WHILE (last-first)>1 DO
	first:=getNextFirstValid(first);
	last:=getNextLastValid(last);
	IF (first<0) OR (last<0) THEN
		RETURN;
	END_IF
END_WHILE

medianValue:=TRUE;
value:=	(inputs[first].input.value+inputs[last].input.value)/2;
END_METHOD

METHOD PRIVATE minValue : BOOL
VAR_INPUT
END_VAR
VAR_OUTPUT
	value:REAL;
END_VAR
VAR
	i:INT;
END_VAR
value:=RNaN();

FOR i:=0 TO arrayMaxIndex DO
	IF isValidInput(inputs[i]) THEN
		IF (FPU.IsRealNaN(value) OR (inputs[i].input.value < value)) THEN
			value:= inputs[i].input.value;
			minValue:=TRUE;
		END_IF
	END_IF
END_FOR
END_METHOD

METHOD PRIVATE compare:bool
VAR_INPUT
	nas1: AnalogItem;
	nas2: AnalogItem;
END_VAR
IF (__ISVALIDREF(nas1.input) AND (NOT __ISVALIDREF (nas2.input))) THEN
	compare:=FALSE;
	RETURN;
END_IF

IF (NOT __ISVALIDREF(nas1.input) AND (__ISVALIDREF (nas2.input))) THEN
	compare:=TRUE;
	RETURN;
END_IF

compare:=FALSE;

IF (__ISVALIDREF(nas1.input) AND __ISVALIDREF (nas2.input)) THEN
	IF 	(nas1.input.interval>=statusAi.normal)AND(nas2.input.interval>=statusAi.normal) THEN
		compare:=nas1.input.value>nas2.input.value;
	ELSE
		compare:=(nas1.input.interval<statusAi.normal)AND(nas2.input.interval>=statusAi.normal)	;			
	END_IF
END_IF
END_METHOD

METHOD sort
VAR_INPUT
END_VAR
VAR
	i,j:INT;
	item:AnalogItem;
	compareResult:BOOL;
END_VAR
FOR i:=1 TO arrayMaxIndex DO
	item:= inputs[i];  
	j:= i - 1;
	compareResult:=compare(nas1:=inputs[j],nas2:=item);
	WHILE (j >= 0) AND (compareResult) DO    
	   	inputs[j + 1]:= inputs[j];
	 	j:=j-1;
	 	IF j>=0 THEN
			compareResult:=compare(nas1:=inputs[j],nas2:=item);
		END_IF
	END_WHILE;
	inputs[j + 1]:= item;
END_FOR
END_METHOD

METHOD PROTECTED writePersistent
VAR_INPUT
END_VAR
SUPER^.writePersistent();
writeValue(value:=FPU.RealToStr(maxDelta),comment:='MAX разброс');
END_METHOD

END_FUNCTION_BLOCK

// lowLevel_ecl/kontroller/mlp/Sources/AoSourceMlp
{attribute 'symbol' := 'none'}
FUNCTION_BLOCK PUBLIC AoSourceMlp EXTENDS AOSource
IMPLEMENTS IMlpSource;
VAR_INPUT
	outLL:REAL:=4000;
	outHl:REAL:=20000;
END_VAR
VAR_OUTPUT
END_VAR
VAR
	elpk:REFERENCE TO Elpk04;
END_VAR

SUPER^();

METHOD setKontroller
VAR_INPUT
	nKontroller	: REFERENCE TO Elpk04;
END_VAR
elpk REF=nKontroller;
END_METHOD

METHOD PROTECTED writeData
VAR_INPUT
	val:REAL;
END_VAR
IF (HL<>LL) THEN
	elpk.Aout_[addr]:=(val-Ll)*(outHl-outLL)/(Hl-Ll)+outLL;
END_IF
END_METHOD

END_FUNCTION_BLOCK

// lowLevel_ecl/kontroller/mlp/Sources/AiFrequenceMlp
{attribute 'symbol' := 'none'}
FUNCTION_BLOCK AiFrequenceMlp EXTENDS AISource
IMPLEMENTS IMlpSource;
VAR_INPUT
	dK:REAL:=1;
	dB:REAL:=0;
END_VAR
VAR_OUTPUT
	{attribute 'symbol' := 'read'}
	k:REAL;
	{attribute 'symbol' := 'read'}
	b:REAL;
END_VAR
VAR
	elpk:REFERENCE TO Elpk04;
	source:AnalogRecalc;
	
	{attribute 'symbol' := 'readwrite'}
	newk:REAL;
	{attribute 'symbol' := 'readwrite'}
	newb:REAL;
END_VAR

SUPER^();

METHOD PROTECTED readPersistent
VAR_INPUT
END_VAR
SUPER^.readPersistent();
K:=FPU.StrToReal(readValue());
B:=FPU.StrToReal(readValue());
END_METHOD

METHOD setKontroller
VAR_INPUT
	nKontroller	: REFERENCE TO Elpk04;
END_VAR
elpk REF=nKontroller;
END_METHOD

METHOD PROTECTED GetData : Real
VAR_INPUT
END_VAR
VAR_OUTPUT
	o_interval:statusAi;
END_VAR
source.input:=elpk.AIn_[addr].val;
source.k:=K;
source.b:=B;
source.h:=histeresis;
source.ap:=aperturFilter;
source.dp:=pikFiler;
source.ds:=exponentialFilter;
source.de:=rassoglasovanie;
source();

GetData:=source.value;

o_interval:=statusAi.normal;
END_METHOD

METHOD PROTECTED writePersistent
VAR_INPUT
END_VAR
SUPER^.writePersistent();
writeValue(value:=FPU.RealToStr(k),comment:='k');
writeValue(value:=FPU.RealToStr(b),comment:='b');
END_METHOD

METHOD PROTECTED setDefaultPersistent:BOOL
VAR_INPUT
END_VAR
SUPER^.setDefaultPersistent();
k:=dK;
b:=dB;
setDefaultPersistent:=TRUE;
END_METHOD

END_FUNCTION_BLOCK

// lowLevel_ecl/kontroller/mlp/Sources/DiSourceMlp
{attribute 'symbol' := 'none'}
FUNCTION_BLOCK DiSourceMlp EXTENDS DISource
IMPLEMENTS IMlpSource;
VAR_INPUT
END_VAR
VAR_OUTPUT
END_VAR
VAR
	elpk:REFERENCE TO Elpk04;
	bitNumber:int;
END_VAR

SUPER^();

METHOD setKontroller
VAR_INPUT
	nKontroller	: REFERENCE TO Elpk04;
END_VAR
elpk REF=nKontroller;
END_METHOD

METHOD PROTECTED getData : word
VAR_INPUT
END_VAR
VAR_OUTPUT
	reliability:WORD;
END_VAR
VAR
	_value:WORD;
	_reliability:BOOL;
END_VAR

_value:=elpk.DIn_[addr].val;
FOR bitNumber:=0 TO 7 DO
	_reliability:=UINT_TO_BOOL(SHR (_value, bitNumber*2) AND 16#2);
	reliability:=reliability OR SHL(BOOL_TO_WORD(_reliability),bitNumber);
	IF _reliability THEN
		getData:=getData OR SHL(SHR (_value, bitNumber*2) AND 16#1,bitNumber);
	END_IF;
END_FOR
END_METHOD

END_FUNCTION_BLOCK

// lowLevel_ecl/kontroller/mlp/Sources/AnalogDiSourceMlp
	{attribute 'symbol' := 'none'}
FUNCTION_BLOCK AnalogDiSourceMlp EXTENDS CustomSource
IMPLEMENTS IMlpSource;
VAR_INPUT
	addr:BYTE;
		 	{attribute 'symbol' := 'readwrite'}
	newTrueLow:REAL;
		 	{attribute 'symbol' := 'readwrite'}
	newTrueHigh:REAL;
		 	{attribute 'symbol' := 'readwrite'}
	newFalseLow:REAL;
		 	{attribute 'symbol' := 'readwrite'}
	newFalseHigh:REAL;
END_VAR
VAR_OUTPUT
	Q:InversableReliableBit;
	{attribute 'symbol' := 'readwrite'}
	value:REAL;
	{attribute 'symbol' := 'readwrite'}
	interval:statusAi;
END_VAR
VAR
	elpk:REFERENCE TO Elpk04;
	source:AnalogRecalc;
		 	{attribute 'symbol' := 'read'}
	trueLow:REAL;
		 	{attribute 'symbol' := 'read'}
	trueHigh:REAL;
		 	{attribute 'symbol' := 'read'}
	falseLow:REAL;
		 	{attribute 'symbol' := 'read'}
	falseHigh:REAL;
END_VAR
VAR CONSTANT
		cmd_changeLimits:WORD:=1;
END_VAR

SUPER^();

IF NOT imit THEN
	source.k:=0.001;
	source.input:=elpk.AIn_[addr].val;
	source();
	value:=source.value;
END_IF

resetCommand();

IF (value>=4) AND (value<=20)  THEN
	IF (value>=falseLow) AND (value<=falseHigh) THEN
		Q.setReliability(TRUE);
		Q.setValue(FALSE);
	ELSIF (value>=trueLow) AND (value<=trueHigh) THEN
		Q.setReliability(TRUE);
		Q.setValue(TRUE);
	ELSE
		Q.setReliability(FALSE);
	END_IF
ELSE
	Q.setReliability(FALSE);
END_IF

METHOD PROTECTED readPersistent
VAR_INPUT
END_VAR
trueLow:=FPU.StrToReal(readValue());
trueHigh:=FPU.StrToReal(readValue());
falseLow:=FPU.StrToReal(readValue());
falseHigh:=FPU.StrToReal(readValue());
END_METHOD

METHOD PROTECTED writePersistent
VAR_INPUT
END_VAR
writeValue(value:=FPU.RealToStr(trueLow),comment:='trueLow');
writeValue(value:=FPU.RealToStr(trueHigh),comment:='trueHigh');
writeValue(value:=FPU.RealToStr(falseLow),comment:='falseLow');
writeValue(value:=FPU.RealToStr(falseHigh),comment:='falseHigh');
END_METHOD

METHOD setLimits
VAR_INPUT
	nFalseLow:REAL;
	nFalseHigh:REAL;
	nTrueLow:REAL;
	nTrueHigh:REAL;

END_VAR
setCmd(nCmd:=cmd_ChangeLimits);
falseLow:=nFalseLow;
falseHigh:=nFalseHigh;
trueLow:=nTrueLow;
trueHigh:=nTrueHigh;

SaveToFile();
END_METHOD

METHOD PROTECTED processCmd;
VAR_INPUT
	cmd:UINT;
	sender:UINT;
	parametr:UINT;
END_VAR
CASE cmd OF
	cmd_changeLimits:setLimits(nFalseLow:=newFalseLow,nFalseHigh:=newFalseHigh,nTrueLow:=newTrueLow,nTrueHigh:=newTrueHigh);
END_CASE
END_METHOD

METHOD setKontroller
VAR_INPUT
	nKontroller	: REFERENCE TO Elpk04;
END_VAR
elpk REF=nKontroller;
END_METHOD

END_FUNCTION_BLOCK

// lowLevel_ecl/kontroller/baseSources/CustomSource
	{attribute 'symbol' := 'none'}
FUNCTION_BLOCK CustomSource EXTENDS BaseIm
IMPLEMENTS ISource
VAR_INPUT

END_VAR
VAR_OUTPUT

END_VAR
VAR
	_imit:BOOL;  
END_VAR

SUPER^();

{attribute 'symbol' := 'none'}
PROPERTY imit : BOOL
SET
_imit:=imit;
END_SET
GET
imit:=_imit;
END_GET
END_PROPERTY

END_FUNCTION_BLOCK

// lowLevel_ecl/kontroller/mlp/Sources/AiSourceMlp
{attribute 'symbol' := 'none'}
FUNCTION_BLOCK AiSourceMlp EXTENDS AISource
IMPLEMENTS IMlpSource;
VAR_INPUT
	inpLL:REAL:=4000;
	inpHl:REAL:=20000;
END_VAR
VAR_OUTPUT
END_VAR
VAR
	elpk:REFERENCE TO Elpk04;
	source:AnalogRecalc;
END_VAR

SUPER^();

METHOD setKontroller
VAR_INPUT
	nKontroller	: REFERENCE TO Elpk04;
END_VAR
elpk REF=nKontroller;
END_METHOD

METHOD PROTECTED GetData : Real
VAR_INPUT
END_VAR
VAR_OUTPUT
	o_interval:statusAi;
END_VAR
source.input:=elpk.AIn_[addr].val;
source.k:=(HL-LL)/(inpHl-inpLL);
source.b:=LL-source.k*inpLL;

source.h:=histeresis;
source.ap:=aperturFilter;
source.dp:=pikFiler;
source.ds:=exponentialFilter;
source.de:=rassoglasovanie;
source();

GetData:=source.value;

IF (NOT (elpk.AIn_[addr].f.0)) OR (NOT (elpk.AIn_[addr].f.2)) OR  (elpk.AIn_[addr].f.1) THEN
	 o_interval:=statusAi.NOTDEFINED;
ELSE
	o_interval:=statusAi.normal;	
END_IF
END_METHOD

END_FUNCTION_BLOCK

// lowLevel_ecl/kontroller/mlp/Sources/DoSourceMlp
{attribute 'symbol' := 'none'}
FUNCTION_BLOCK DoSourceMlp EXTENDS DOSource
IMPLEMENTS IMlpSource;
VAR_INPUT
END_VAR
VAR_OUTPUT
END_VAR
VAR
	elpk:REFERENCE TO Elpk04;
END_VAR

SUPER^();

METHOD setKontroller
VAR_INPUT
	nKontroller	: REFERENCE TO Elpk04;
END_VAR
elpk REF=nKontroller;
END_METHOD

METHOD writeData
VAR_INPUT
	value:WORD;
END_VAR
elpk.Dout_[addr]:=value;
END_METHOD

END_FUNCTION_BLOCK

// lowLevel_ecl/im/extensions/ExtNarabotka
	{attribute 'symbol' := 'none'}
FUNCTION_BLOCK ExtNarabotka EXTENDS BaseObject
VAR_INPUT
	saveInterval:TIME:=T#30S;
END_VAR
VAR_OUTPUT
	{attribute 'symbol' := 'read'}
	narabotka:UDINT;	
END_VAR
VAR
END_VAR
VAR
	timer:RTC;	
	saveTimer:TON;
END_VAR

SUPER^();
timer();

IF timer.Q THEN
	narabotka:=DT_TO_UDINT( timer.CDT);
END_IF

saveTimer(IN:=TRUE,PT:=saveInterval);
IF saveTimer.Q THEN
	SaveToFile();
	saveTimer(IN:=FALSE);
END_IF

METHOD PROTECTED readPersistent
VAR_INPUT
END_VAR
narabotka:=STRING_TO_UDINT(readValue());
END_METHOD

METHOD PUBLIC reset
VAR_INPUT
END_VAR
timer.PDT:=UINT_TO_DT(0);
IF timer.EN THEN
	timer(EN:=FALSE);
	timer(EN:=TRUE);
END_IF
narabotka:=0;
END_METHOD

METHOD PUBLIC start
VAR_INPUT
END_VAR
timer.PDT:=UDINT_TO_DT(narabotka);
timer.EN:=TRUE;
END_METHOD

PROPERTY PUBLIC started : Bool
GET
started:=timer.Q;
END_GET
SET
IF started then
	IF NOT timer.Q THEN
		start();
	END_IF
ELSE
	IF timer.Q THEN
		stop();
	END_IF
END_IF
END_SET
END_PROPERTY

METHOD PUBLIC stop
VAR_INPUT
END_VAR
timer.EN:=FALSE;
SaveToFile();
END_METHOD

METHOD PROTECTED writePersistent
VAR_INPUT
END_VAR
writeValue(value:= UDINT_TO_STRING(narabotka),'Наработка');
END_METHOD

END_FUNCTION_BLOCK

// lowLevel_ecl/im/Mokveld/Mokveld
	{attribute 'symbol' := 'none'}
FUNCTION_BLOCK Mokveld EXTENDS BaseIm
VAR_INPUT
	inPosition:REFERENCE TO AISource;
	inAssignment:REFERENCE TO AOSource;
	
	dMaxOpenSpeed:REAL:=RNaN();
	dMaxCloseSpeed:REAL:=RNaN();
	
	maxPositionMismatch:REAL:=RNaN();
	posotionnMismatchDelay:TIME:=T#5S;
	
	openPosition:REAL:=95;
	closePosition:REAL:=5;
	
		{attribute 'symbol' := 'readwrite'}
	newTarget:REAL;
END_VAR
VAR_OUTPUT
	{attribute 'symbol' := 'read'}
	position:REAL;
	{attribute 'symbol' := 'read'}
	target:REAL;	

	Assignment:REAL;	
	
	onStatus:statusDualInput;
	
	positionMismatch:BOOL;
END_VAR
VAR
	maxOpenSpeed:REAL;
	maxCloseSpeed:REAL;
	lastCallTimer:Ton:=(pt:=T#1H);
	posotionErrorTimer:TON;
END_VAR
VAR CONSTANT
	cmd_setTarget:WORD:=1;
END_VAR
VAR_TEMP
	delta:REAL:=RNaN();
END_VAR

SUPER^();

IF __ISVALIDREF(inPosition) THEN
	position:=inPosition.value;
	
	IF inPosition.interval>=statusAi.normal THEN
		IF (NOT FPU.IsRealNaN(maxPositionMismatch)) AND __ISVALIDREF(inAssignment) THEN
			posotionErrorTimer(IN:= rABS(inAssignment.Value-inPosition.value)>maxPositionMismatch,PT:=posotionnMismatchDelay);
			PositionMismatch:=posotionErrorTimer.Q;
		END_IF	
		onStatus:=calcOnStatus();
	ELSE
		onStatus:=statusDualInput.STATUS_ERROR;
		posotionErrorTimer(IN:=FALSE);
	END_IF
ELSE
	IF __ISVALIDREF(inAssignment) THEN
		position:=inAssignment.Value;
		onStatus:=calcOnStatus();			
	END_IF
END_IF

IF __ISVALIDREF(inAssignment) THEN
	inAssignment.DisableOpcControl();

	lastCallTimer();
	IF (target>inAssignment.Value) THEN 
		IF NOT FPU.IsRealNaN(maxOpenSpeed) THEN 
			delta:=maxOpenSpeed*(TIME_TO_REAL(lastCallTimer.ET)/1000);
		END_IF;
	ELSE
		IF NOT FPU.IsRealNaN(maxCloseSpeed) THEN
			delta:=-maxCloseSpeed*(TIME_TO_REAL(lastCallTimer.ET)/1000);
		END_IF	
	END_IF
	lastCallTimer(in:=FALSE);
	lastCallTimer(in:=TRUE);
		
	IF (NOT FPU.IsRealNaN(delta)) AND (ABS(delta)<ABS(inAssignment.Value-target)) THEN
		Assignment:=inAssignment.Value+delta;
	ELSE
		Assignment:=target;	
	END_IF
	
	inAssignment.setValue(nValue:=Assignment);
END_IF

METHOD PROTECTED calcOnStatus: statusDualInput
VAR_INPUT
END_VAR
IF (position<closePosition) THEN
	calcOnStatus:=statusDualInput.STATUS_OFF;
ELSIF (position>openPosition) THEN
	calcOnStatus:=statusDualInput.STATUS_ON;
ELSE
	calcOnStatus:=statusDualInput.STATUS_TRANSITIONAL;
END_IF
END_METHOD

METHOD PRIVATE cmdSetTarget
VAR_INPUT
	nTarget:REAL;
END_VAR
setCmd(nCmd:=cmd_setTarget);
setTarget(nTarget:=nTarget);
resetCommand();
END_METHOD

METHOD PROTECTED processCmd;
VAR_INPUT
	cmd:UINT;
	sender:UINT;
	parametr:UINT;
END_VAR
SUPER^.processCmd(cmd,sender,parametr);
CASE cmd OF
	cmd_setTarget: cmdSetTarget(nTarget:=newTarget);
END_CASE
END_METHOD

METHOD PROTECTED readPersistent
VAR_INPUT
END_VAR
SUPER^.readPersistent();
maxOpenSpeed:=FPU.StrToReal(readValue());
maxCloseSpeed:=FPU.StrToReal(readValue());
openPosition:=FPU.StrToReal(readValue());
closePosition:=FPU.StrToReal(readValue());
END_METHOD

METHOD PROTECTED setDefaultPersistent:BOOL
VAR_INPUT
END_VAR
SUPER^.setDefaultPersistent();
maxOpenSpeed:=dMaxOpenSpeed;
maxCloseSpeed:=dMaxCloseSpeed;
setDefaultPersistent:=TRUE;
END_METHOD

METHOD PUBLIC setTarget
VAR_INPUT
	nTarget:REAL;
END_VAR
target:=nTarget;
END_METHOD

METHOD PUBLIC writeImStatus
VAR_INPUT
END_VAR
statusSet.setBits(0,2,onStatus);
statusSet.setBit(3,positionMismatch);
END_METHOD

METHOD PROTECTED writePersistent
VAR_INPUT
END_VAR
SUPER^.writePersistent();
writeValue(value:=FPU.RealToStr(maxOpenSpeed),comment:='maxOpenSpeed');
writeValue(value:=FPU.RealToStr(maxCloseSpeed),comment:='maxCloseSpeed');
writeValue(value:=FPU.RealToStr(openPosition),comment:='openPosition');
writeValue(value:=FPU.RealToStr(closePosition),comment:='closePosition');
END_METHOD

END_FUNCTION_BLOCK

// REZERV1/ADDCRC16
FUNCTION ADDCRC16 : WORD
VAR_INPUT
	X:BYTE;
	_CRC16T:WORD;
END_VAR
VAR
	CRC16_B:BOOL;
	I:INT;
	T:WORD;
END_VAR

FOR I:=1 TO 8 DO
	
	T:=BYTE_TO_WORD(X) XOR _CRC16T;
	IF (T AND 16#1) = 1// если нечетное, то = true
		THEN
		CRC16_B:=TRUE;
		ELSE
		CRC16_B:=FALSE;
	END_IF

	_CRC16T:= SHR(_CRC16T, 1);
	X:= SHR(X,1);
	IF CRC16_B THEN _CRC16T:=_CRC16T XOR 16#A001; END_IF;

END_FOR
ADDCRC16:=_CRC16T;

END_FUNCTION

// REZERV1/COM_Rd
FUNCTION_BLOCK COM_Rd
VAR CONSTANT
	Buff_size12:INT:=12;
	Byte_send12:UINT:=12;
END_VAR
VAR_INPUT
	PilaK_O:WORD;
	StatusK_O:WORD;
	ReadyK_O:WORD;
END_VAR
VAR_IN_OUT
//	IndexCmd:INT:=-1;// команда на запись переменной Index с экрана
	IndexCmd:INT;// команда на запись переменной Index с экрана - инициализировать сверху
	Cnt0:INT:=0;// счетчик правильных заголовков пакета: 0x81 + (длина=12) 
	Cnt100:INT:=0;// счетчик ошибок длины пакета 
	Cnt101:INT:=0;// счетчик ошибок признака начала пакета 0x81
	Cnt102:INT:=0;// счетчик ошибок CRC16
	Cnt3:INT:=0;// для ошибок Write
	Cnt21:INT:=0;// для ошибок Read
	Cnt22:INT:=0;// для ошибок Read
	Cnt23:INT:=0;// для ошибок Read
	Cnt24:INT:=0;// для ошибок Read
	Cnt25:INT:=0;// для ошибок Read
	Cnt26:INT:=0;// для ошибок Read
	Cnt27:INT:=0;// для ошибок Read
	Cnt28:INT:=0;// для ошибок Read
	Cnt29:INT:=0;// для ошибок Read
	Cnt30:INT:=0;// для ошибок Read
	Cnt31:INT:=0;// для ошибок Read
	Cnt32:INT:=0;// для ошибок Read
END_VAR
VAR_OUTPUT
	// принятое из соседнего
	PilaFromK:WORD;
	StatusFromK:WORD;
	ReadyFromK:WORD;
	ErrorCOM_Mess1, ErrorCOM_Mess2:WSTRING;
	
END_VAR
VAR
	Index:INT:=0;
//	IndexCmd:INT:=-1;// команда на запись переменной Index с экрана
	I1, I2, I3, I4 :INT;// переменные временного использования
	PP1, PP2, PP3, PP4, PP5 : RTS_IEC_RESULT;
///	H1 : RTS_IEC_HANDLE;// pointer to byte
///	S1 : Com_Settings;
///	S1ex : Com_SettingsEX;

{attribute 'displaymode':='hex'} 
	Buff : ARRAY[1..Buff_size12] OF BYTE;
{attribute 'displaymode':='hex'} 
	Buff2 : ARRAY[1..Buff_size12] OF BYTE;
//{attribute 'displaymode':='hex'} 
//	Buff22 : ARRAY[1..Buff_size12] OF BYTE;
//	ErrorCOM_Mess1, ErrorCOM_Mess2:WSTRING;
	
	
	WW1, WW2, WW3,WW4,WW5,WW6,WW7,WW8,WW9,WW10,WW10a,WW10b:UDINT;
	WW11,WW12,WW13,WW14,WW15,WW16,WW17,WW18,WW19,WW20,WW21,WW22:UDINT;
//////////////////////////////////////////////////////////////

	PacketOK_Other:BYTE:=0;
//	PacketOK_CntOther:INT;

	// вычисленная КС для передачи
	CRC16O:WORD;
	// вычисленная КС для приема
	CRC16_1, CRC16_2:WORD;


	PP21, PP22, PP23, PP24, PP25, PP26, PP27, PP28, PP29, PP30 : RTS_IEC_RESULT;
	//Cnt21,Cnt22,Cnt23,Cnt24,Cnt25,Cnt26,Cnt27,Cnt28,Cnt29,Cnt30:INT:=0;// для ошибок Read
	PP31, PP32, PP33, PP34, PP35, PP36, PP37, PP38, PP39, PP40 : RTS_IEC_RESULT;
//	Cnt31,Cnt32,
Cnt33,Cnt34,Cnt35,Cnt36,Cnt37,Cnt38,Cnt39,Cnt40:INT:=0;// для ошибок Read
	Cnt4:INT:=0;// для ошибок Read
	
	PP41, PP42, PP43, PP44, PP45 : RTS_IEC_RESULT;
	Cnt41:INT:=0;// для ошибок Read
	Cnt42:INT:=0;// для ошибок Read
	Cnt43:INT:=0;// для ошибок Read
	Cnt44:INT:=0;// для ошибок Read
	
END_VAR

// только чтение

CASE Index OF
0:



IF (H1=RTS_INVALID_HANDLE)OR(H1=0)
	THEN
//	Index:=3;// закрыть порт и ждать	
	RETURN;// выйти - ждать пока появится хандл
END_IF
 



(*	
// установить параметры COM-портов
S1.sPort:= 1;//=1 - Com1
S1.byStopBits:= Sys_ONESTOPBIT;//=1
S1.byParity:= Sys_NOPARITY;// =0
S1.ulBaudrate:= SYS_BR_19200;	//SYS_BR_9600; SYS_BR_19200;  SYS_BR_115200
S1.ulTimeout:= 0;
S1.ulBufferSize:=0;
///H1:= SysCom.SysComOpen(SYS_COMPORT1, ADR(PP1));
H1:= SysComOpen2(ADR(S1), ADR(S1ex), ADR(PP1));
*)
Index:=21;
/////Index:=100;


Index:=41;




IF H1=RTS_INVALID_HANDLE
	THEN
	Index:=3;// закрыть порт и ждать	
	RETURN;
END_IF


2:
	CASE IndexCmd OF
	0..3:// есть что-то для записи
		Index:=IndexCmd;
		IndexCmd:=-1;// сбросить команду
		RETURN;
	ELSE
		IndexCmd:=-1;// сбросить команду
	END_CASE

	FOR I1:=1 TO Buff_size12 DO
		Buff2[I1]:= 0;	// очистить буфер для нового чтения 
	END_FOR

	
	
	FOR I1:=1 TO Buff_size12+5 DO
	WW11:=SysComRead(H1, ADR(Buff2[1]), 1, {SYS_INFINITE}50, ADR(PP41));// Start_Packet
	IF PP41 <> 0
		THEN
		 Cnt41:=Cnt41+1;
//		 CONTINUE;
//		 RETURN;
//		PP2:= SysComPurge(H1);
	END_IF// ошибки
	IF (Buff2[1] = 16#81){AND(Buff2[2] = 12} 
		THEN
			I2:=I1;
		 	EXIT;
	END_IF
	IF I1 >= Buff_size12
		THEN
		PP2:= SysComPurge(H1);
	END_IF
	END_FOR

	
	// читать пакеты соседа
//	WW11:=SysComRead(H1, ADR(Buff2[1]), 1, {SYS_INFINITE}120, ADR(PP4));// Start_Packet
//	IF PP4 <> 0	THEN Cnt4:=Cnt4+1; END_IF// ошибки
	IF Buff2[1] = 16#81
		THEN
		// читать пакеты соседа
		WW12:=SysComRead(H1, ADR(Buff2[2]), 1, {SYS_INFINITE}10, ADR(PP4));//Len_Packet
		IF PP4 <> 0	THEN Cnt4:=Cnt4+1; RETURN; END_IF// ошибки
		IF Buff2[2] = Byte_send12
			THEN
			// читать пакеты соседа
			WW13:=SysComRead(H1, ADR(Buff2[3]), 1, {SYS_INFINITE}10, ADR(PP4));// PacketOK_Other
			IF PP4 <> 0	THEN Cnt4:=Cnt4+1; RETURN; END_IF// ошибки
			// читать пакеты соседа
			WW14:=SysComRead(H1, ADR(Buff2[4]), 1, {SYS_INFINITE}10, ADR(PP4));// Rezerv
			IF PP4 <> 0	THEN Cnt4:=Cnt4+1; RETURN; END_IF// ошибки
			// читать пакеты соседа
			WW15:=SysComRead(H1, ADR(Buff2[5]), 1, {SYS_INFINITE}10, ADR(PP4));// PilaK1_O - ст
			IF PP4 <> 0	THEN Cnt4:=Cnt4+1; RETURN; END_IF// ошибки
			// читать пакеты соседа
			WW16:=SysComRead(H1, ADR(Buff2[6]), 1, {SYS_INFINITE}10, ADR(PP4));// PilaK1_O - мл
			IF PP4 <> 0	THEN Cnt4:=Cnt4+1; RETURN; END_IF// ошибки
			// читать пакеты соседа
			WW17:=SysComRead(H1, ADR(Buff2[7]), 1, {SYS_INFINITE}10, ADR(PP4));// StatusK1_O - ст
			IF PP4 <> 0	THEN Cnt4:=Cnt4+1; RETURN; END_IF// ошибки
			// читать пакеты соседа
			WW18:=SysComRead(H1, ADR(Buff2[8]), 1, {SYS_INFINITE}10, ADR(PP4));// StatusK1_O - мл
			IF PP4 <> 0	THEN Cnt4:=Cnt4+1; RETURN; END_IF// ошибки
			// читать пакеты соседа
			WW19:=SysComRead(H1, ADR(Buff2[9]), 1, {SYS_INFINITE}10, ADR(PP4));// ReadyK1_O - ст
			IF PP4 <> 0	THEN Cnt4:=Cnt4+1; RETURN; END_IF// ошибки
			// читать пакеты соседа
			WW20:=SysComRead(H1, ADR(Buff2[10]), 1, {SYS_INFINITE}10, ADR(PP4));// ReadyK1_O - мл
			IF PP4 <> 0	THEN Cnt4:=Cnt4+1; RETURN; END_IF// ошибки
			// читать пакеты соседа
			WW21:=SysComRead(H1, ADR(Buff2[11]), 1, {SYS_INFINITE}10, ADR(PP4));// KS
			IF PP4 <> 0	THEN Cnt4:=Cnt4+1; RETURN; END_IF// ошибки
			// читать пакеты соседа
			WW22:=SysComRead(H1, ADR(Buff2[12]), 1, {SYS_INFINITE}10, ADR(PP4));//KS
			IF PP4 <> 0	THEN Cnt4:=Cnt4+1; RETURN; END_IF// ошибки

//			PilaFromK:=  (SHL(Buff2[5],8) AND 16#FF) OR (Buff2[6] AND 16#FF);
//			StatusFromK:=(SHL(Buff2[7],8) AND 16#FF) OR (Buff2[8] AND 16#FF);
//			ReadyFromK:= (SHL(Buff2[9],8) AND 16#FF) OR (Buff2[10] AND 16#FF);
//			CRC16:= (SHL(Buff2[11],8) AND 16#FF) OR (Buff2[12] AND 16#FF);

			// восстановить CRC, принятую в пакете из соседнего
			CRC16_1:= Buff2[11];// ст.байт КС
			CRC16_1:= SHL(CRC16_1,8);
			CRC16_1:= CRC16_1 AND 16#FF00;
			CRC16_1:= CRC16_1 OR Buff2[12];// мл.байт КС
			// подсчитать CRC принятого пакета
			CRC16_2:=0;
			FOR I1:=1 TO Buff_size12-2 DO
//			FOR I1:=1 TO Buff_size12 DO
				CRC16_2:=ADDCRC16(Buff2[I1], CRC16_2);
			END_FOR
			// проверить КС

			IF CRC16_1=CRC16_2
//			IF CRC16_2=0
			THEN
				PilaFromK:= Buff2[5];
				PilaFromK:= SHL(PilaFromK,8);
				PilaFromK:= PilaFromK AND 16#FF00;
				PilaFromK:= PilaFromK OR Buff2[6];
			
				StatusFromK:= Buff2[7];
				StatusFromK:= SHL(StatusFromK,8);
				StatusFromK:= StatusFromK AND 16#FF00;
				StatusFromK:= StatusFromK OR Buff2[8];
			
				ReadyFromK:= Buff2[9];
				ReadyFromK:= SHL(ReadyFromK,8);
				ReadyFromK:= ReadyFromK AND 16#FF00;
				ReadyFromK:= ReadyFromK OR Buff2[10];
			
				PacketOK_Other:=16#55;// признак правильного пакета при приеме пакета от соседа
			ELSE
				Cnt102:=Cnt102+1;
				PacketOK_Other:=0;// признак ошибки при приеме пакета от соседа
//				SysComPurge(H1);// сбросить буфера
			END_IF 
			ELSE
			Cnt100:=Cnt100+1;
			PacketOK_Other:=0;// признак ошибки при приеме пакета от соседа
//			SysComPurge(H1);// сбросить буфера
		END_IF  
		ELSE
			Cnt101:=Cnt101+1;
			PacketOK_Other:=0;// признак ошибки при приеме пакета от соседа
//			SysComPurge(H1);// сбросить буфера
	END_IF

	Index:=1;//?????
			PP2:= SysComPurge(H1);


3:
	PP5:=SysComClose(H1);
	// здесь можно сформировать признак ошибки СОМ-порта "ComOpen ERROR"
	ErrorCOM_Mess1:="Com1 Open Error";
	Index:=10;
	
4:
	PP5:=SysComClose(H1);
	// здесь можно сформировать признак ошибки СОМ-порта "ComPurge ERROR"
	ErrorCOM_Mess1:="Com1 Purge Error";
//	Index:=1;// возобновить работу СОМ
	Index:=10;

5:
	PP5:=SysComClose(H1);
	// здесь можно сформировать признак ошибки СОМ-порта "ComWrite ERROR"
	ErrorCOM_Mess1:="Com1 Write Error";
	Index:=10;// возобновить работу СОМ
	
6:
	PP5:=SysComClose(H1);
	// здесь можно сформировать признак ошибки СОМ-порта "ComRead ERROR"
	ErrorCOM_Mess1:="Com1 Read Error";
	Index:=10;// возобновить работу СОМ

7:
	// здесь можно сформировать признак ошибки СОМ-порта "Packet ERROR"
	//	ошибка целостности пакета
	ErrorCOM_Mess1:="Com1 Packet Error";
	Index:=10;// возобновить работу СОМ

10:
	// здесь можно сформировать признак ошибки СОМ-порта
	ErrorCOM_Mess2:="Com1 Can't Open or Close";



21:
	CASE IndexCmd OF
	0..3:// есть что-то для записи
		Index:=IndexCmd;
		IndexCmd:=-1;// сбросить команду
		RETURN;
	ELSE
		IndexCmd:=-1;// сбросить команду
	END_CASE

	FOR I1:=1 TO Buff_size12 DO
		Buff2[I1]:= 0;	// очистить буфер для нового чтения 
	END_FOR

	FOR I1:=1 TO Buff_size12+5 DO
	WW11:=SysComRead(H1, ADR(Buff2[1]), 1, {SYS_INFINITE}150, ADR(PP21));// Start_Packet
	IF PP21 <> 0
		THEN
		 Cnt21:=Cnt21+1;
//		 CONTINUE;
//		Index:=1;
		Index:=31;
//		PP2:= SysComPurge(H1);
		 RETURN;
	END_IF// ошибки

	IF (Buff2[1] = 16#81){AND(Buff2[2] = 12} 
		THEN
	WW12:=SysComRead(H1, ADR(Buff2[2]), 1, {SYS_INFINITE}20, ADR(PP22));// Start_Packet
	IF PP22 <> 0
		THEN
		 Cnt22:=Cnt22+1;
//		 CONTINUE;
//		Index:=1;
		Index:=31;
		 RETURN;
//		PP2:= SysComPurge(H1);
	END_IF// ошибки

	IF {(Buff2[1] = 16#81)AND}(Buff2[2] = Byte_send12) 
		THEN
		 	Cnt0:=Cnt0+1;
			I2:=I1;
			Index:=22;
			 RETURN;

	ELSE
			Cnt100:=Cnt100+1;
			PacketOK_Other:=0;// признак ошибки при приеме пакета от соседа
//			SysComPurge(H1);// сбросить буфера
	END_IF
	ELSE
			Cnt101:=Cnt101+1;
			PacketOK_Other:=0;// признак ошибки при приеме пакета от соседа
//			SysComPurge(H1);// сбросить буфера
	END_IF

	END_FOR

	Index:=31;
///////			SysComPurge(H1);// сбросить буфера

	
22:	

			// читать пакеты соседа
			WW13:=SysComRead(H1, ADR(Buff2[3]), 1, {SYS_INFINITE}10, ADR(PP23));// PacketOK_Other
			IF PP23 <> 0	THEN Cnt23:=Cnt23+1; {RETURN;} END_IF// ошибки
			// читать пакеты соседа
			WW14:=SysComRead(H1, ADR(Buff2[4]), 1, {SYS_INFINITE}10, ADR(PP24));// Rezerv
			IF PP24 <> 0	THEN Cnt24:=Cnt24+1; {RETURN;} END_IF// ошибки
			// читать пакеты соседа
			WW15:=SysComRead(H1, ADR(Buff2[5]), 1, {SYS_INFINITE}10, ADR(PP25));// PilaK1_O - ст
			IF PP25 <> 0	THEN Cnt25:=Cnt25+1; {RETURN;} END_IF// ошибки
			// читать пакеты соседа
			WW16:=SysComRead(H1, ADR(Buff2[6]), 1, {SYS_INFINITE}10, ADR(PP26));// PilaK1_O - мл
			IF PP26 <> 0	THEN Cnt26:=Cnt26+1; {RETURN;} END_IF// ошибки
			// читать пакеты соседа
			WW17:=SysComRead(H1, ADR(Buff2[7]), 1, {SYS_INFINITE}10, ADR(PP27));// StatusK1_O - ст
			IF PP27 <> 0	THEN Cnt27:=Cnt27+1; {RETURN;} END_IF// ошибки
			// читать пакеты соседа
			WW18:=SysComRead(H1, ADR(Buff2[8]), 1, {SYS_INFINITE}10, ADR(PP28));// StatusK1_O - мл
			IF PP28 <> 0	THEN Cnt28:=Cnt28+1; {RETURN;} END_IF// ошибки
			// читать пакеты соседа
			WW19:=SysComRead(H1, ADR(Buff2[9]), 1, {SYS_INFINITE}20, ADR(PP29));// ReadyK1_O - ст
			IF PP29 <> 0	THEN Cnt29:=Cnt29+1; {RETURN;} END_IF// ошибки
			// читать пакеты соседа
			WW20:=SysComRead(H1, ADR(Buff2[10]), 1, {SYS_INFINITE}20, ADR(PP30));// ReadyK1_O - мл
			IF PP30 <> 0	THEN Cnt30:=Cnt30+1; {RETURN;} END_IF// ошибки
			// читать пакеты соседа
			WW21:=SysComRead(H1, ADR(Buff2[11]), 1, {SYS_INFINITE}30, ADR(PP31));// KS
			IF PP31 <> 0	THEN Cnt31:=Cnt31+1; {RETURN;} END_IF// ошибки
			// читать пакеты соседа
			WW22:=SysComRead(H1, ADR(Buff2[12]), 1, {SYS_INFINITE}30, ADR(PP32));//KS
			IF PP32 <> 0	THEN Cnt32:=Cnt32+1; {RETURN;} END_IF// ошибки

			// восстановить CRC, принятую в пакете из соседнего
			CRC16_1:= Buff2[11];// ст.байт КС
			CRC16_1:= SHL(CRC16_1,8);
			CRC16_1:= CRC16_1 AND 16#FF00;
			CRC16_1:= CRC16_1 OR Buff2[12];// мл.байт КС
			// подсчитать CRC принятого пакета
			CRC16_2:=0;
			FOR I1:=1 TO Buff_size12-2 DO
//			FOR I1:=1 TO Buff_size12 DO
				CRC16_2:=ADDCRC16(Buff2[I1], CRC16_2);
			END_FOR
			// проверить КС
			
			IF CRC16_1=CRC16_2
//			IF CRC16_2=0
			THEN
				PilaFromK:= Buff2[5];
				PilaFromK:= SHL(PilaFromK,8);
				PilaFromK:= PilaFromK AND 16#FF00;
				PilaFromK:= PilaFromK OR Buff2[6];
			
				StatusFromK:= Buff2[7];
				StatusFromK:= SHL(StatusFromK,8);
				StatusFromK:= StatusFromK AND 16#FF00;
				StatusFromK:= StatusFromK OR Buff2[8];
			
				ReadyFromK:= Buff2[9];
				ReadyFromK:= SHL(ReadyFromK,8);
				ReadyFromK:= ReadyFromK AND 16#FF00;
				ReadyFromK:= ReadyFromK OR Buff2[10];
			
				PacketOK_Other:=16#55;// признак правильного пакета при приеме пакета от соседа
			ELSE
				Cnt102:=Cnt102+1;
				PacketOK_Other:=0;// признак ошибки при приеме пакета от соседа
//				SysComPurge(H1);// сбросить буфера
			END_IF 
			
	Index:=21;
	
	
31:
	Index:=21;
32:
	Index:=21;


	
	
	
100:
	CASE IndexCmd OF
	0..3:// есть что-то для записи
		Index:=IndexCmd;
		IndexCmd:=-1;// сбросить команду
		RETURN;
	ELSE
		IndexCmd:=-1;// сбросить команду
	END_CASE

	FOR I1:=1 TO Buff_size12 DO
		Buff2[I1]:= 0;	// очистить буфер для нового чтения 
	END_FOR
   	Index:=101;
	
	
101:
	CASE IndexCmd OF
	0..3:// есть что-то для записи
		Index:=IndexCmd;
		IndexCmd:=-1;// сбросить команду
		RETURN;
	ELSE
		IndexCmd:=-1;// сбросить команду
	END_CASE
	
	WW11:=SysComRead(H1, ADR(Buff2[1]), 1, {SYS_INFINITE}150, ADR(PP21));// Start_Packet
	IF PP21 <> 0
		THEN
		Cnt21:=Cnt21+1;
    	Index:=100;
		RETURN;
	END_IF// ошибки
	IF (Buff2[1] = 16#81){AND(Buff2[2] = 12} 
		THEN
    	Index:=102;
		ELSE
		Cnt101:=Cnt101+1;
		PacketOK_Other:=0;// признак ошибки при приеме пакета от соседа
	END_IF// ошибки

102:
	CASE IndexCmd OF
	0..3:// есть что-то для записи
		Index:=IndexCmd;
		IndexCmd:=-1;// сбросить команду
		RETURN;
	ELSE
		IndexCmd:=-1;// сбросить команду
	END_CASE
	
	WW12:=SysComRead(H1, ADR(Buff2[2]), 1, {SYS_INFINITE}150, ADR(PP22));// Start_Packet
	IF PP22 <> 0
		THEN
		Cnt22:=Cnt22+1;
    	Index:=100;
		RETURN;
	END_IF// ошибки
	IF (Buff2[2] = 16#0C) 
		THEN
    	Index:=103;
		ELSE
		Cnt100:=Cnt100+1;
		PacketOK_Other:=0;// признак ошибки при приеме пакета от соседа
	END_IF// ошибки
103:
	// читать пакеты соседа
	WW13:=SysComRead(H1, ADR(Buff2[3]), 1, {SYS_INFINITE}10, ADR(PP23));// PacketOK_Other
	IF PP23 <> 0	
		THEN
		Cnt23:=Cnt23+1;
		RETURN;
	END_IF// ошибки
	IF WW13 <> 0	
		THEN
    	Index:=104;
		ELSE
		RETURN;
	END_IF// ошибки
104:
	// читать пакеты соседа
	WW14:=SysComRead(H1, ADR(Buff2[4]), 1, {SYS_INFINITE}10, ADR(PP24));// PacketOK_Other
	IF PP24 <> 0	
		THEN
		Cnt24:=Cnt24+1;
		RETURN;
	END_IF// ошибки
	IF WW14 <> 0	
		THEN
    	Index:=105;
		ELSE
		RETURN;
	END_IF// ошибки
105:
	// читать пакеты соседа
	WW15:=SysComRead(H1, ADR(Buff2[5]), 1, {SYS_INFINITE}10, ADR(PP25));// PacketOK_Other
	IF PP25 <> 0	
		THEN
		Cnt25:=Cnt25+1;
		RETURN;
	END_IF// ошибки
	IF WW15 <> 0	
		THEN
    	Index:=106;
		ELSE
		RETURN;
	END_IF// ошибки
	
106:
	// читать пакеты соседа
	WW16:=SysComRead(H1, ADR(Buff2[6]), 1, {SYS_INFINITE}10, ADR(PP26));// PacketOK_Other
	IF PP26 <> 0	
		THEN
		Cnt26:=Cnt26+1;
		RETURN;
	END_IF// ошибки
	IF WW16 <> 0	
		THEN
    	Index:=107;
		ELSE
		RETURN;
	END_IF// ошибки
107:
	// читать пакеты соседа
	WW17:=SysComRead(H1, ADR(Buff2[7]), 1, {SYS_INFINITE}10, ADR(PP27));// PacketOK_Other
	IF PP27 <> 0	
		THEN
		Cnt27:=Cnt27+1;
		RETURN;
	END_IF// ошибки
	IF WW17 <> 0	
		THEN
    	Index:=108;
		ELSE
		RETURN;
	END_IF// ошибки
108:
	// читать пакеты соседа
	WW18:=SysComRead(H1, ADR(Buff2[8]), 1, {SYS_INFINITE}10, ADR(PP28));// PacketOK_Other
	IF PP28 <> 0	
		THEN
		Cnt28:=Cnt28+1;
		RETURN;
	END_IF// ошибки
	IF WW18 <> 0	
		THEN
    	Index:=109;
		ELSE
		RETURN;
	END_IF// ошибки
109:
	// читать пакеты соседа
	WW19:=SysComRead(H1, ADR(Buff2[9]), 1, {SYS_INFINITE}10, ADR(PP29));// PacketOK_Other
	IF PP29 <> 0	
		THEN
		Cnt29:=Cnt29+1;
		RETURN;
	END_IF// ошибки
	IF WW19 <> 0	
		THEN
    	Index:=110;
		ELSE
		RETURN;
	END_IF// ошибки
110:
	// читать пакеты соседа
	WW20:=SysComRead(H1, ADR(Buff2[10]), 1, {SYS_INFINITE}10, ADR(PP30));// PacketOK_Other
	IF PP30 <> 0	
		THEN
		Cnt30:=Cnt30+1;
		RETURN;
	END_IF// ошибки
	IF WW20 <> 0	
		THEN
    	Index:=111;
		ELSE
		RETURN;
	END_IF// ошибки
111:
	// читать пакеты соседа
	WW21:=SysComRead(H1, ADR(Buff2[11]), 1, {SYS_INFINITE}10, ADR(PP31));// PacketOK_Other
	IF PP31 <> 0	
		THEN
		Cnt31:=Cnt31+1;
		RETURN;
	END_IF// ошибки
	IF WW21 <> 0	
		THEN
    	Index:=112;
		ELSE
		RETURN;
	END_IF// ошибки
112:
	// читать пакеты соседа
	WW22:=SysComRead(H1, ADR(Buff2[12]), 1, {SYS_INFINITE}10, ADR(PP32));// PacketOK_Other
	IF PP32 <> 0	
		THEN
		Cnt32:=Cnt32+1;
		RETURN;
	END_IF// ошибки
	IF WW22 <> 0	
		THEN
///    	Index:=113;
		ELSE
		RETURN;
	END_IF// ошибки
	
	

	
			// восстановить CRC, принятую в пакете из соседнего
			CRC16_1:= Buff2[11];// ст.байт КС
			CRC16_1:= SHL(CRC16_1,8);
			CRC16_1:= CRC16_1 AND 16#FF00;
			CRC16_1:= CRC16_1 OR Buff2[12];// мл.байт КС
			// подсчитать CRC принятого пакета
			CRC16_2:=0;
			FOR I1:=1 TO Buff_size12-2 DO
				CRC16_2:=ADDCRC16(Buff2[I1], CRC16_2);
			END_FOR
			// проверить КС
			
			IF CRC16_1=CRC16_2
			THEN
				PilaFromK:= Buff2[5];
				PilaFromK:= SHL(PilaFromK,8);
				PilaFromK:= PilaFromK AND 16#FF00;
				PilaFromK:= PilaFromK OR Buff2[6];
			
				StatusFromK:= Buff2[7];
				StatusFromK:= SHL(StatusFromK,8);
				StatusFromK:= StatusFromK AND 16#FF00;
				StatusFromK:= StatusFromK OR Buff2[8];
			
				ReadyFromK:= Buff2[9];
				ReadyFromK:= SHL(ReadyFromK,8);
				ReadyFromK:= ReadyFromK AND 16#FF00;
				ReadyFromK:= ReadyFromK OR Buff2[10];
			
				PacketOK_Other:=16#55;// признак правильного пакета при приеме пакета от соседа
			ELSE
				Cnt102:=Cnt102+1;
				PacketOK_Other:=0;// признак ошибки при приеме пакета от соседа
//				SysComPurge(H1);// сбросить буфера
			END_IF 
	
	
	
		Index:=100;



41:
	CASE IndexCmd OF
	0..3:// есть что-то для записи
		Index:=IndexCmd;
		IndexCmd:=-1;// сбросить команду
		RETURN;
	ELSE
		IndexCmd:=-1;// сбросить команду
	END_CASE

	FOR I1:=1 TO Buff_size12 DO
		Buff2[I1]:= 0;	// очистить буфер для нового чтения 
	END_FOR


///	FOR I1:=1 TO Buff_size12 DO
	
	
	WW11:=SysComRead(H1, ADR(Buff2[1]), 1, {SYS_INFINITE}10, ADR(PP21));// Start_Packet
	IF PP21 <> 0	
		THEN// есть ошибка таймаута
		Cnt21:=Cnt21+1;
		RETURN;
//		CONTINUE;
	END_IF// ошибки
	IF (Buff2[1] <> 16#81) OR (WW11=0)	
		THEN
		Cnt31:=Cnt31+1;
		RETURN;
///		CONTINUE;
	END_IF// ошибки

	WW12:=SysComRead(H1, ADR(Buff2[2]), 1, {SYS_INFINITE}10, ADR(PP22));// Start_Packet
	IF PP22 <> 0	
		THEN
		Cnt22:=Cnt22+1;
		RETURN;
//		CONTINUE;
	END_IF// ошибки
	IF (Buff2[2] <> 16#0C) OR (WW12=0)	
		THEN
		Cnt32:=Cnt32+1;
		RETURN;
///		CONTINUE;
	END_IF// ошибки
	Index:=42;
///		EXIT;////////////////////
///	END_FOR

42:	
	
	
	WW13:=SysComRead(H1, ADR(Buff2[3]), 10, {SYS_INFINITE}{100}50, ADR(PP23));// Start_Packet
	IF (PP23 <> 0) OR (WW13<>10)	
		THEN
		Cnt23:=Cnt23+1;
		RETURN;
	END_IF// ошибки

			// восстановить CRC, принятую в пакете из соседнего
			CRC16_1:= Buff2[11];// ст.байт КС
			CRC16_1:= SHL(CRC16_1,8);
			CRC16_1:= CRC16_1 AND 16#FF00;
			CRC16_1:= CRC16_1 OR Buff2[12];// мл.байт КС
			// подсчитать CRC принятого пакета
			CRC16_2:=0;
			FOR I1:=1 TO Buff_size12-2 DO
				CRC16_2:=ADDCRC16(Buff2[I1], CRC16_2);
			END_FOR
			// проверить КС
			
			IF CRC16_1=CRC16_2
			THEN
				PilaFromK:= Buff2[5];
				PilaFromK:= SHL(PilaFromK,8);
				PilaFromK:= PilaFromK AND 16#FF00;
				PilaFromK:= PilaFromK OR Buff2[6];
			
				StatusFromK:= Buff2[7];
				StatusFromK:= SHL(StatusFromK,8);
				StatusFromK:= StatusFromK AND 16#FF00;
				StatusFromK:= StatusFromK OR Buff2[8];
			
				ReadyFromK:= Buff2[9];
				ReadyFromK:= SHL(ReadyFromK,8);
				ReadyFromK:= ReadyFromK AND 16#FF00;
				ReadyFromK:= ReadyFromK OR Buff2[10];
			
				PacketOK_Other:=16#55;// признак правильного пакета при приеме пакета от соседа
				Cnt0:=Cnt0+1;
			ELSE
				Cnt102:=Cnt102+1;
				PacketOK_Other:=0;// признак ошибки при приеме пакета от соседа
//				SysComPurge(H1);// сбросить буфера
			END_IF 

	

	Index:=41;
	

150:
		PP2:= SysComPurge(H1);
///	Index:=21;
////	Index:=100;
	Index:=41;


	
END_CASE

END_FUNCTION_BLOCK

// REZERV1/COM1
FUNCTION_BLOCK COM1
VAR CONSTANT
	Buff_size12:INT:=12;
	Byte_send12:UINT:=12;
END_VAR
VAR_INPUT
	PilaK_O:WORD;
	StatusK_O:WORD;
	ReadyK_O:WORD;
END_VAR
VAR_IN_OUT
//	IndexCmd:INT:=-1;// команда на запись переменной Index с экрана
	IndexCmd:INT;// команда на запись переменной Index с экрана - инициализировать сверху
	Cnt0:INT:=0;// счетчик правильных заголовков пакета: 0x81 + (длина=12) 
	Cnt100:INT:=0;// счетчик ошибок длины пакета 
	Cnt101:INT:=0;// счетчик ошибок признака начала пакета 0x81
	Cnt102:INT:=0;// счетчик ошибок CRC16
	Cnt3:INT:=0;// для ошибок Write
	Cnt21:INT:=0;// для ошибок Read
	Cnt22:INT:=0;// для ошибок Read
	Cnt23:INT:=0;// для ошибок Read
	Cnt24:INT:=0;// для ошибок Read
	Cnt25:INT:=0;// для ошибок Read
	Cnt26:INT:=0;// для ошибок Read
	Cnt27:INT:=0;// для ошибок Read
	Cnt28:INT:=0;// для ошибок Read
	Cnt29:INT:=0;// для ошибок Read
	Cnt30:INT:=0;// для ошибок Read
	Cnt31:INT:=0;// для ошибок Read
	Cnt32:INT:=0;// для ошибок Read
END_VAR
VAR_OUTPUT
	// принятое из соседнего
	PilaFromK:WORD;
	StatusFromK:WORD;
	ReadyFromK:WORD;
	ErrorCOM_Mess1, ErrorCOM_Mess2:WSTRING;
	
END_VAR
VAR
	Index:INT:=0;
//	IndexCmd:INT:=-1;// команда на запись переменной Index с экрана
	I1, I2, I3, I4 :INT;// переменные временного использования
	PP1, PP2, PP3, PP4, PP5 : RTS_IEC_RESULT;
	H1 : RTS_IEC_HANDLE;// pointer to byte
	S1 : Com_Settings;
	S1ex : Com_SettingsEX;

{attribute 'displaymode':='hex'} 
	Buff : ARRAY[1..Buff_size12] OF BYTE;
{attribute 'displaymode':='hex'} 
	Buff2 : ARRAY[1..Buff_size12] OF BYTE;
//{attribute 'displaymode':='hex'} 
//	Buff22 : ARRAY[1..Buff_size12] OF BYTE;
//	ErrorCOM_Mess1, ErrorCOM_Mess2:WSTRING;
	
	
	WW1, WW2, WW3,WW4,WW5,WW6,WW7,WW8,WW9,WW10,WW10a,WW10b:UDINT;
	WW11,WW12,WW13,WW14,WW15,WW16,WW17,WW18,WW19,WW20,WW21,WW22:UDINT;
//////////////////////////////////////////////////////////////

	PacketOK_Other:BYTE:=0;
//	PacketOK_CntOther:INT;

	// вычисленная КС для передачи
	CRC16O:WORD;
	// вычисленная КС для приема
	CRC16_1, CRC16_2:WORD;


	PP21, PP22, PP23, PP24, PP25, PP26, PP27, PP28, PP29, PP30 : RTS_IEC_RESULT;
	//Cnt21,Cnt22,Cnt23,Cnt24,Cnt25,Cnt26,Cnt27,Cnt28,Cnt29,Cnt30:INT:=0;// для ошибок Read
	PP31, PP32, PP33, PP34, PP35, PP36, PP37, PP38, PP39, PP40 : RTS_IEC_RESULT;
//	Cnt31,Cnt32,
Cnt33,Cnt34,Cnt35,Cnt36,Cnt37,Cnt38,Cnt39,Cnt40:INT:=0;// для ошибок Read
	Cnt4:INT:=0;// для ошибок Read
	
	PP41, PP42, PP43, PP44, PP45 : RTS_IEC_RESULT;
	Cnt41:INT:=0;// для ошибок Read
	Cnt42:INT:=0;// для ошибок Read
	Cnt43:INT:=0;// для ошибок Read
	Cnt44:INT:=0;// для ошибок Read
	
END_VAR

CASE Index OF
0:	
// установить параметры COM-портов
S1.sPort:= 1;//=1 - Com1
S1.byStopBits:= Sys_ONESTOPBIT;//=1
S1.byParity:= Sys_NOPARITY;// =0
S1.ulBaudrate:= SYS_BR_19200;	//SYS_BR_9600; SYS_BR_19200;  SYS_BR_115200
S1.ulTimeout:= 0;
S1.ulBufferSize:=0;
///H1:= SysCom.SysComOpen(SYS_COMPORT1, ADR(PP1));
H1:= SysComOpen2(ADR(S1), ADR(S1ex), ADR(PP1));

Index:=1;

IF H1=RTS_INVALID_HANDLE
	THEN
	Index:=3;// закрыть порт и ждать	
	RETURN;
END_IF

1:
	CASE IndexCmd OF
	0..3:// есть что-то для записи с экрана
		Index:=IndexCmd;
		IndexCmd:=-1;// сбросить команду
		RETURN;
	ELSE
		IndexCmd:=-1;// сбросить команду
	END_CASE 
	
	// очистить строки ошибок
	ErrorCOM_Mess1:=ErrorCOM_Mess2:="";
	// очистить буфера приема/передачи
	FOR I1:=1 TO Buff_size12 DO
		Buff[I1]:= 0;
	END_FOR
	// заполнить буфер передачи
	Buff[1]:= UINT_TO_BYTE(16#81);// признак начала пакета
	Buff[2]:= UINT_TO_BYTE(Byte_send12);// размер пакета
	Buff[3]:= PacketOK_Other;// вернуть признак правильного приема пакета
	Buff[4]:= 0;// резерв
	// слова - вперед головой !!!
	Buff[5]:= UINT_TO_BYTE(SHR(PilaK_O,8) AND 16#FF);// ст байт
	Buff[6]:= UINT_TO_BYTE(PilaK_O AND 16#FF);// мл байт
	Buff[7]:= UINT_TO_BYTE(SHR(StatusK_O,8) AND 16#FF);// ст байт
	Buff[8]:= UINT_TO_BYTE(StatusK_O AND 16#FF);// мл байт
	Buff[9]:= UINT_TO_BYTE(SHR(ReadyK_O,8) AND 16#FF);// ст байт
	Buff[10]:=UINT_TO_BYTE(ReadyK_O AND 16#FF);// мл байт

///////////////////////////////////////////////////
//	Buff[3]:=3; Buff[4]:=4; Buff[5]:=5; Buff[6]:=6; Buff[7]:=7; Buff[8]:=8; Buff[9]:=9; Buff[10]:=10;
///////////////////////////////////////////////////
	
	
	// подсчитать КС
	CRC16O:=0;
	FOR I1:=1 TO Buff_size12-2 DO
		CRC16O:=ADDCRC16(Buff[I1], CRC16O);
	END_FOR
	Buff[11]:=WORD_TO_BYTE(SHR(CRC16O,8) AND 16#FF);// ст байт
	Buff[12]:=WORD_TO_BYTE(CRC16O AND 16#FF);// мл байт
//	Buff[11]:= 0;// KS
//	Buff[12]:= 0;// KS
  
	// послать буфер в порт 
	WW1:=SysComWrite(H1, ADR(Buff), Byte_send12{10}, {SYS_INFINITE}50, ADR(PP3));
(*
	WW1:=SysComWrite(H1, ADR(Buff[1]), 1, {SYS_INFINITE}10, ADR(PP3));
	WW2:=SysComWrite(H1, ADR(Buff[2]), 1, {SYS_INFINITE}10, ADR(PP3));
	WW3:=SysComWrite(H1, ADR(Buff[3]), 1, {SYS_INFINITE}10, ADR(PP3));
	WW4:=SysComWrite(H1, ADR(Buff[4]), 1, {SYS_INFINITE}10, ADR(PP3));
	WW5:=SysComWrite(H1, ADR(Buff[5]), 1, {SYS_INFINITE}10, ADR(PP3));
	WW6:=SysComWrite(H1, ADR(Buff[6]), 1, {SYS_INFINITE}10, ADR(PP3));
	WW7:=SysComWrite(H1, ADR(Buff[7]), 1, {SYS_INFINITE}10, ADR(PP3));
	WW8:=SysComWrite(H1, ADR(Buff[8]), 1, {SYS_INFINITE}10, ADR(PP3));
	WW9:=SysComWrite(H1, ADR(Buff[9]), 1, {SYS_INFINITE}10, ADR(PP3));
	WW10:=SysComWrite(H1, ADR(Buff[10]), 1, {SYS_INFINITE}10, ADR(PP3));
	WW10a:=SysComWrite(H1, ADR(Buff[11]), 1, {SYS_INFINITE}10, ADR(PP3));
	WW10b:=SysComWrite(H1, ADR(Buff[12]), 1, {SYS_INFINITE}10, ADR(PP3));
*)
	IF PP3=5// таймаут
		THEN// ошибки
		PP2:= SysComPurge(H1);
		Cnt3:=Cnt3+1;
	END_IF
	
//	Index:=2;
//	Index:=21;
	Index:=32;

2:
	CASE IndexCmd OF
	0..3:// есть что-то для записи
		Index:=IndexCmd;
		IndexCmd:=-1;// сбросить команду
		RETURN;
	ELSE
		IndexCmd:=-1;// сбросить команду
	END_CASE

	FOR I1:=1 TO Buff_size12 DO
		Buff2[I1]:= 0;	// очистить буфер для нового чтения 
	END_FOR

	
	
	FOR I1:=1 TO Buff_size12+5 DO
	WW11:=SysComRead(H1, ADR(Buff2[1]), 1, {SYS_INFINITE}50, ADR(PP41));// Start_Packet
	IF PP41 <> 0
		THEN
		 Cnt41:=Cnt41+1;
//		 CONTINUE;
//		 RETURN;
//		PP2:= SysComPurge(H1);
	END_IF// ошибки
	IF (Buff2[1] = 16#81){AND(Buff2[2] = 12} 
		THEN
			I2:=I1;
		 	EXIT;
	END_IF
	IF I1 >= Buff_size12
		THEN
		PP2:= SysComPurge(H1);
	END_IF
	END_FOR

	
	// читать пакеты соседа
//	WW11:=SysComRead(H1, ADR(Buff2[1]), 1, {SYS_INFINITE}120, ADR(PP4));// Start_Packet
//	IF PP4 <> 0	THEN Cnt4:=Cnt4+1; END_IF// ошибки
	IF Buff2[1] = 16#81
		THEN
		// читать пакеты соседа
		WW12:=SysComRead(H1, ADR(Buff2[2]), 1, {SYS_INFINITE}10, ADR(PP4));//Len_Packet
		IF PP4 <> 0	THEN Cnt4:=Cnt4+1; RETURN; END_IF// ошибки
		IF Buff2[2] = Byte_send12
			THEN
			// читать пакеты соседа
			WW13:=SysComRead(H1, ADR(Buff2[3]), 1, {SYS_INFINITE}10, ADR(PP4));// PacketOK_Other
			IF PP4 <> 0	THEN Cnt4:=Cnt4+1; RETURN; END_IF// ошибки
			// читать пакеты соседа
			WW14:=SysComRead(H1, ADR(Buff2[4]), 1, {SYS_INFINITE}10, ADR(PP4));// Rezerv
			IF PP4 <> 0	THEN Cnt4:=Cnt4+1; RETURN; END_IF// ошибки
			// читать пакеты соседа
			WW15:=SysComRead(H1, ADR(Buff2[5]), 1, {SYS_INFINITE}10, ADR(PP4));// PilaK1_O - ст
			IF PP4 <> 0	THEN Cnt4:=Cnt4+1; RETURN; END_IF// ошибки
			// читать пакеты соседа
			WW16:=SysComRead(H1, ADR(Buff2[6]), 1, {SYS_INFINITE}10, ADR(PP4));// PilaK1_O - мл
			IF PP4 <> 0	THEN Cnt4:=Cnt4+1; RETURN; END_IF// ошибки
			// читать пакеты соседа
			WW17:=SysComRead(H1, ADR(Buff2[7]), 1, {SYS_INFINITE}10, ADR(PP4));// StatusK1_O - ст
			IF PP4 <> 0	THEN Cnt4:=Cnt4+1; RETURN; END_IF// ошибки
			// читать пакеты соседа
			WW18:=SysComRead(H1, ADR(Buff2[8]), 1, {SYS_INFINITE}10, ADR(PP4));// StatusK1_O - мл
			IF PP4 <> 0	THEN Cnt4:=Cnt4+1; RETURN; END_IF// ошибки
			// читать пакеты соседа
			WW19:=SysComRead(H1, ADR(Buff2[9]), 1, {SYS_INFINITE}10, ADR(PP4));// ReadyK1_O - ст
			IF PP4 <> 0	THEN Cnt4:=Cnt4+1; RETURN; END_IF// ошибки
			// читать пакеты соседа
			WW20:=SysComRead(H1, ADR(Buff2[10]), 1, {SYS_INFINITE}10, ADR(PP4));// ReadyK1_O - мл
			IF PP4 <> 0	THEN Cnt4:=Cnt4+1; RETURN; END_IF// ошибки
			// читать пакеты соседа
			WW21:=SysComRead(H1, ADR(Buff2[11]), 1, {SYS_INFINITE}10, ADR(PP4));// KS
			IF PP4 <> 0	THEN Cnt4:=Cnt4+1; RETURN; END_IF// ошибки
			// читать пакеты соседа
			WW22:=SysComRead(H1, ADR(Buff2[12]), 1, {SYS_INFINITE}10, ADR(PP4));//KS
			IF PP4 <> 0	THEN Cnt4:=Cnt4+1; RETURN; END_IF// ошибки

//			PilaFromK:=  (SHL(Buff2[5],8) AND 16#FF) OR (Buff2[6] AND 16#FF);
//			StatusFromK:=(SHL(Buff2[7],8) AND 16#FF) OR (Buff2[8] AND 16#FF);
//			ReadyFromK:= (SHL(Buff2[9],8) AND 16#FF) OR (Buff2[10] AND 16#FF);
//			CRC16:= (SHL(Buff2[11],8) AND 16#FF) OR (Buff2[12] AND 16#FF);

			// восстановить CRC, принятую в пакете из соседнего
			CRC16_1:= Buff2[11];// ст.байт КС
			CRC16_1:= SHL(CRC16_1,8);
			CRC16_1:= CRC16_1 AND 16#FF00;
			CRC16_1:= CRC16_1 OR Buff2[12];// мл.байт КС
			// подсчитать CRC принятого пакета
			CRC16_2:=0;
			FOR I1:=1 TO Buff_size12-2 DO
//			FOR I1:=1 TO Buff_size12 DO
				CRC16_2:=ADDCRC16(Buff2[I1], CRC16_2);
			END_FOR
			// проверить КС

			IF CRC16_1=CRC16_2
//			IF CRC16_2=0
			THEN
				PilaFromK:= Buff2[5];
				PilaFromK:= SHL(PilaFromK,8);
				PilaFromK:= PilaFromK AND 16#FF00;
				PilaFromK:= PilaFromK OR Buff2[6];
			
				StatusFromK:= Buff2[7];
				StatusFromK:= SHL(StatusFromK,8);
				StatusFromK:= StatusFromK AND 16#FF00;
				StatusFromK:= StatusFromK OR Buff2[8];
			
				ReadyFromK:= Buff2[9];
				ReadyFromK:= SHL(ReadyFromK,8);
				ReadyFromK:= ReadyFromK AND 16#FF00;
				ReadyFromK:= ReadyFromK OR Buff2[10];
			
				PacketOK_Other:=16#55;// признак правильного пакета при приеме пакета от соседа
			ELSE
				Cnt102:=Cnt102+1;
				PacketOK_Other:=0;// признак ошибки при приеме пакета от соседа
//				SysComPurge(H1);// сбросить буфера
			END_IF 
			ELSE
			Cnt100:=Cnt100+1;
			PacketOK_Other:=0;// признак ошибки при приеме пакета от соседа
//			SysComPurge(H1);// сбросить буфера
		END_IF  
		ELSE
			Cnt101:=Cnt101+1;
			PacketOK_Other:=0;// признак ошибки при приеме пакета от соседа
//			SysComPurge(H1);// сбросить буфера
	END_IF

	Index:=1;
			PP2:= SysComPurge(H1);


3:
	PP5:=SysComClose(H1);
	// здесь можно сформировать признак ошибки СОМ-порта "ComOpen ERROR"
	ErrorCOM_Mess1:="Com1 Open Error";
	Index:=10;
	
4:
	PP5:=SysComClose(H1);
	// здесь можно сформировать признак ошибки СОМ-порта "ComPurge ERROR"
	ErrorCOM_Mess1:="Com1 Purge Error";
//	Index:=1;// возобновить работу СОМ
	Index:=10;

5:
	PP5:=SysComClose(H1);
	// здесь можно сформировать признак ошибки СОМ-порта "ComWrite ERROR"
	ErrorCOM_Mess1:="Com1 Write Error";
	Index:=1;// возобновить работу СОМ
	
6:
	PP5:=SysComClose(H1);
	// здесь можно сформировать признак ошибки СОМ-порта "ComRead ERROR"
	ErrorCOM_Mess1:="Com1 Read Error";
	Index:=1;// возобновить работу СОМ

7:
	// здесь можно сформировать признак ошибки СОМ-порта "Packet ERROR"
	//	ошибка целостности пакета
	ErrorCOM_Mess1:="Com1 Packet Error";
	Index:=1;// возобновить работу СОМ

10:
	// здесь можно сформировать признак ошибки СОМ-порта
	ErrorCOM_Mess2:="Com1 Can't Open or Close";



21:
	CASE IndexCmd OF
	0..3:// есть что-то для записи
		Index:=IndexCmd;
		IndexCmd:=-1;// сбросить команду
		RETURN;
	ELSE
		IndexCmd:=-1;// сбросить команду
	END_CASE

	FOR I1:=1 TO Buff_size12 DO
		Buff2[I1]:= 0;	// очистить буфер для нового чтения 
	END_FOR

	FOR I1:=1 TO Buff_size12+5 DO
	WW11:=SysComRead(H1, ADR(Buff2[1]), 1, {SYS_INFINITE}150, ADR(PP21));// Start_Packet
	IF PP21 <> 0
		THEN
		 Cnt21:=Cnt21+1;
//		 CONTINUE;
//		Index:=1;
		Index:=31;
//		PP2:= SysComPurge(H1);
		 RETURN;
	END_IF// ошибки

	IF (Buff2[1] = 16#81){AND(Buff2[2] = 12} 
		THEN
	WW12:=SysComRead(H1, ADR(Buff2[2]), 1, {SYS_INFINITE}20, ADR(PP22));// Start_Packet
	IF PP22 <> 0
		THEN
		 Cnt22:=Cnt22+1;
//		 CONTINUE;
//		Index:=1;
		Index:=31;
		 RETURN;
//		PP2:= SysComPurge(H1);
	END_IF// ошибки

	IF {(Buff2[1] = 16#81)AND}(Buff2[2] = Byte_send12) 
		THEN
		 	Cnt0:=Cnt0+1;
			I2:=I1;
			Index:=22;
			 RETURN;
//		 	EXIT;
	ELSE
			Cnt100:=Cnt100+1;
			PacketOK_Other:=0;// признак ошибки при приеме пакета от соседа
//			SysComPurge(H1);// сбросить буфера
	END_IF
	ELSE
			Cnt101:=Cnt101+1;
			PacketOK_Other:=0;// признак ошибки при приеме пакета от соседа
//			SysComPurge(H1);// сбросить буфера
	END_IF

	END_FOR

	Index:=31;
////			SysComPurge(H1);// сбросить буфера

	
22:	

			// читать пакеты соседа
			WW13:=SysComRead(H1, ADR(Buff2[3]), 1, {SYS_INFINITE}10, ADR(PP23));// PacketOK_Other
			IF PP23 <> 0	THEN Cnt23:=Cnt23+1; {RETURN;} END_IF// ошибки
			// читать пакеты соседа
			WW14:=SysComRead(H1, ADR(Buff2[4]), 1, {SYS_INFINITE}10, ADR(PP24));// Rezerv
			IF PP24 <> 0	THEN Cnt24:=Cnt24+1; {RETURN;} END_IF// ошибки
			// читать пакеты соседа
			WW15:=SysComRead(H1, ADR(Buff2[5]), 1, {SYS_INFINITE}10, ADR(PP25));// PilaK1_O - ст
			IF PP25 <> 0	THEN Cnt25:=Cnt25+1; {RETURN;} END_IF// ошибки
			// читать пакеты соседа
			WW16:=SysComRead(H1, ADR(Buff2[6]), 1, {SYS_INFINITE}10, ADR(PP26));// PilaK1_O - мл
			IF PP26 <> 0	THEN Cnt26:=Cnt26+1; {RETURN;} END_IF// ошибки
			// читать пакеты соседа
			WW17:=SysComRead(H1, ADR(Buff2[7]), 1, {SYS_INFINITE}10, ADR(PP27));// StatusK1_O - ст
			IF PP27 <> 0	THEN Cnt27:=Cnt27+1; {RETURN;} END_IF// ошибки
			// читать пакеты соседа
			WW18:=SysComRead(H1, ADR(Buff2[8]), 1, {SYS_INFINITE}10, ADR(PP28));// StatusK1_O - мл
			IF PP28 <> 0	THEN Cnt28:=Cnt28+1; {RETURN;} END_IF// ошибки
			// читать пакеты соседа
			WW19:=SysComRead(H1, ADR(Buff2[9]), 1, {SYS_INFINITE}10, ADR(PP29));// ReadyK1_O - ст
			IF PP29 <> 0	THEN Cnt29:=Cnt29+1; {RETURN;} END_IF// ошибки
			// читать пакеты соседа
			WW20:=SysComRead(H1, ADR(Buff2[10]), 1, {SYS_INFINITE}10, ADR(PP30));// ReadyK1_O - мл
			IF PP30 <> 0	THEN Cnt30:=Cnt30+1; {RETURN;} END_IF// ошибки
			// читать пакеты соседа
			WW21:=SysComRead(H1, ADR(Buff2[11]), 1, {SYS_INFINITE}20, ADR(PP31));// KS
			IF PP31 <> 0	THEN Cnt31:=Cnt31+1; {RETURN;} END_IF// ошибки
			// читать пакеты соседа
			WW22:=SysComRead(H1, ADR(Buff2[12]), 1, {SYS_INFINITE}20, ADR(PP32));//KS
			IF PP32 <> 0	THEN Cnt32:=Cnt32+1; {RETURN;} END_IF// ошибки

			// восстановить CRC, принятую в пакете из соседнего
			CRC16_1:= Buff2[11];// ст.байт КС
			CRC16_1:= SHL(CRC16_1,8);
			CRC16_1:= CRC16_1 AND 16#FF00;
			CRC16_1:= CRC16_1 OR Buff2[12];// мл.байт КС
			// подсчитать CRC принятого пакета
			CRC16_2:=0;
			FOR I1:=1 TO Buff_size12-2 DO
//			FOR I1:=1 TO Buff_size12 DO
				CRC16_2:=ADDCRC16(Buff2[I1], CRC16_2);
			END_FOR
			// проверить КС
			
			IF CRC16_1=CRC16_2
//			IF CRC16_2=0
			THEN
				PilaFromK:= Buff2[5];
				PilaFromK:= SHL(PilaFromK,8);
				PilaFromK:= PilaFromK AND 16#FF00;
				PilaFromK:= PilaFromK OR Buff2[6];
			
				StatusFromK:= Buff2[7];
				StatusFromK:= SHL(StatusFromK,8);
				StatusFromK:= StatusFromK AND 16#FF00;
				StatusFromK:= StatusFromK OR Buff2[8];
			
				ReadyFromK:= Buff2[9];
				ReadyFromK:= SHL(ReadyFromK,8);
				ReadyFromK:= ReadyFromK AND 16#FF00;
				ReadyFromK:= ReadyFromK OR Buff2[10];
			
				PacketOK_Other:=16#55;// признак правильного пакета при приеме пакета от соседа
			ELSE
				Cnt102:=Cnt102+1;
				PacketOK_Other:=0;// признак ошибки при приеме пакета от соседа
//				SysComPurge(H1);// сбросить буфера
			END_IF 
			
	Index:=1;
	
	
31:
	Index:=1;
32:
	Index:=21;



150:
		PP2:= SysComPurge(H1);
	Index:=1;


	
END_CASE

END_FUNCTION_BLOCK

// REZERV1/COM_Wr
FUNCTION_BLOCK COM_Wr
VAR CONSTANT
	Buff_size12:INT:=12;
	Byte_send12:UINT:=12;
END_VAR
VAR_INPUT
	PilaK_O:WORD;
	StatusK_O:WORD;
	ReadyK_O:WORD;
END_VAR
VAR_IN_OUT
//	IndexCmd:INT:=-1;// команда на запись переменной Index с экрана
	IndexCmd:INT;// команда на запись переменной Index с экрана - инициализировать сверху
//	Cnt0:INT:=0;// счетчик правильных заголовков пакета: 0x81 + (длина=12) 
//	Cnt100:INT:=0;// счетчик ошибок длины пакета 
//	Cnt101:INT:=0;// счетчик ошибок признака начала пакета 0x81
//	Cnt102:INT:=0;// счетчик ошибок CRC16
	Cnt3:INT:=0;// для ошибок Write
//	Cnt21:INT:=0;// для ошибок Read
//	Cnt22:INT:=0;// для ошибок Read
//	Cnt23:INT:=0;// для ошибок Read
//	Cnt24:INT:=0;// для ошибок Read
//	Cnt25:INT:=0;// для ошибок Read
//	Cnt26:INT:=0;// для ошибок Read
//	Cnt27:INT:=0;// для ошибок Read
//	Cnt28:INT:=0;// для ошибок Read
//	Cnt29:INT:=0;// для ошибок Read
//	Cnt30:INT:=0;// для ошибок Read
//	Cnt31:INT:=0;// для ошибок Read
//	Cnt32:INT:=0;// для ошибок Read
END_VAR
VAR_OUTPUT
	// принятое из соседнего
//	PilaFromK:WORD;
//	StatusFromK:WORD;
//	ReadyFromK:WORD;
	ErrorCOM_Mess1, ErrorCOM_Mess2:WSTRING;
END_VAR
VAR
	Index:INT:=0;
//	IndexCmd:INT:=-1;// команда на запись переменной Index с экрана
	I1, I2, I3, I4 :INT;// переменные временного использования
	PP1, PP2, PP3, PP4, PP5 : RTS_IEC_RESULT;
///	H1 : RTS_IEC_HANDLE;// pointer to byte
///	S1 : Com_Settings;
///	S1ex : Com_SettingsEX;

{attribute 'displaymode':='hex'} 
	Buff : ARRAY[1..Buff_size12] OF BYTE;
{attribute 'displaymode':='hex'} 
	Buff2 : ARRAY[1..Buff_size12] OF BYTE;
//{attribute 'displaymode':='hex'} 
//	Buff22 : ARRAY[1..Buff_size12] OF BYTE;
//	ErrorCOM_Mess1, ErrorCOM_Mess2:WSTRING;
	
	
	WW1, WW2, WW3,WW4,WW5,WW6,WW7,WW8,WW9,WW10,WW10a,WW10b:UDINT;
	WW11,WW12,WW13,WW14,WW15,WW16,WW17,WW18,WW19,WW20,WW21,WW22:UDINT;
//////////////////////////////////////////////////////////////

	PacketOK_Other:BYTE:=0;
//	PacketOK_CntOther:INT;

	// вычисленная КС для передачи
	CRC16O:WORD;
	// вычисленная КС для приема
	CRC16_1, CRC16_2:WORD;


	PP21, PP22, PP23, PP24, PP25, PP26, PP27, PP28, PP29, PP30 : RTS_IEC_RESULT;
	//Cnt21,Cnt22,Cnt23,Cnt24,Cnt25,Cnt26,Cnt27,Cnt28,Cnt29,Cnt30:INT:=0;// для ошибок Read
	PP31, PP32, PP33, PP34, PP35, PP36, PP37, PP38, PP39, PP40 : RTS_IEC_RESULT;
//	Cnt31,Cnt32,
Cnt33,Cnt34,Cnt35,Cnt36,Cnt37,Cnt38,Cnt39,Cnt40:INT:=0;// для ошибок Read
	Cnt4:INT:=0;// для ошибок Read
	
	PP41, PP42, PP43, PP44, PP45 : RTS_IEC_RESULT;
	Cnt41:INT:=0;// для ошибок Read
	Cnt42:INT:=0;// для ошибок Read
	Cnt43:INT:=0;// для ошибок Read
	Cnt44:INT:=0;// для ошибок Read
	
END_VAR

// только запись

CASE Index OF
0:	
// установить параметры COM-портов
S1.sPort:= 1;//=1 - Com1
S1.byStopBits:= Sys_ONESTOPBIT;//=1
S1.byParity:= Sys_NOPARITY;// =0
S1.ulBaudrate:= SYS_BR_9600;	//SYS_BR_9600; SYS_BR_19200;  SYS_BR_115200
//S1.ulBaudrate:= SYS_BR_19200;	//SYS_BR_9600; SYS_BR_19200;  SYS_BR_115200

///S1.ulTimeout:= 0;
///S1.ulBufferSize:=0;

S1.ulTimeout:= 300;
S1.ulBufferSize:=16;


///H1:= SysCom.SysComOpen(SYS_COMPORT1, ADR(PP1));
H1:= SysComOpen2(ADR(S1), ADR(S1ex), ADR(PP1));

Index:=1;

IF H1=RTS_INVALID_HANDLE
	THEN
	Index:=3;// закрыть порт и ждать	
	RETURN;
END_IF

1:
	CASE IndexCmd OF
	0..3:// есть что-то для записи с экрана
		Index:=IndexCmd;
		IndexCmd:=-1;// сбросить команду
		RETURN;
	ELSE
		IndexCmd:=-1;// сбросить команду
	END_CASE 
	
	// очистить строки ошибок
	ErrorCOM_Mess1:=ErrorCOM_Mess2:="";
	// очистить буфера приема/передачи
	FOR I1:=1 TO Buff_size12 DO
		Buff[I1]:= 0;
	END_FOR
	// заполнить буфер передачи
	Buff[1]:= UINT_TO_BYTE(16#81);// признак начала пакета
	Buff[2]:= UINT_TO_BYTE(Byte_send12);// размер пакета
	Buff[3]:= PacketOK_Other;// вернуть признак правильного приема пакета
	Buff[4]:= 0;// резерв
	// слова - вперед головой !!!
	Buff[5]:= UINT_TO_BYTE(SHR(PilaK_O,8) AND 16#FF);// ст байт
	Buff[6]:= UINT_TO_BYTE(PilaK_O AND 16#FF);// мл байт
	Buff[7]:= UINT_TO_BYTE(SHR(StatusK_O,8) AND 16#FF);// ст байт
	Buff[8]:= UINT_TO_BYTE(StatusK_O AND 16#FF);// мл байт
	Buff[9]:= UINT_TO_BYTE(SHR(ReadyK_O,8) AND 16#FF);// ст байт
	Buff[10]:=UINT_TO_BYTE(ReadyK_O AND 16#FF);// мл байт

///////////////////////////////////////////////////
//	Buff[3]:=3; Buff[4]:=4; Buff[5]:=5; Buff[6]:=6; Buff[7]:=7; Buff[8]:=8; Buff[9]:=9; Buff[10]:=10;
///////////////////////////////////////////////////
	
	
	// подсчитать КС
	CRC16O:=0;
	FOR I1:=1 TO Buff_size12-2 DO
		CRC16O:=ADDCRC16(Buff[I1], CRC16O);
	END_FOR
	Buff[11]:=WORD_TO_BYTE(SHR(CRC16O,8) AND 16#FF);// ст байт
	Buff[12]:=WORD_TO_BYTE(CRC16O AND 16#FF);// мл байт
//	Buff[11]:= 0;// KS
//	Buff[12]:= 0;// KS
  
	// послать буфер в порт 
	WW1:=SysComWrite(H1, ADR(Buff), Byte_send12{10}, {SYS_INFINITE}{50}150, ADR(PP3));
(*
	WW1:=SysComWrite(H1, ADR(Buff[1]), 1, {SYS_INFINITE}10, ADR(PP3));
	WW2:=SysComWrite(H1, ADR(Buff[2]), 1, {SYS_INFINITE}10, ADR(PP3));
	WW3:=SysComWrite(H1, ADR(Buff[3]), 1, {SYS_INFINITE}10, ADR(PP3));
	WW4:=SysComWrite(H1, ADR(Buff[4]), 1, {SYS_INFINITE}10, ADR(PP3));
	WW5:=SysComWrite(H1, ADR(Buff[5]), 1, {SYS_INFINITE}10, ADR(PP3));
	WW6:=SysComWrite(H1, ADR(Buff[6]), 1, {SYS_INFINITE}10, ADR(PP3));
	WW7:=SysComWrite(H1, ADR(Buff[7]), 1, {SYS_INFINITE}10, ADR(PP3));
	WW8:=SysComWrite(H1, ADR(Buff[8]), 1, {SYS_INFINITE}10, ADR(PP3));
	WW9:=SysComWrite(H1, ADR(Buff[9]), 1, {SYS_INFINITE}10, ADR(PP3));
	WW10:=SysComWrite(H1, ADR(Buff[10]), 1, {SYS_INFINITE}10, ADR(PP3));
	WW10a:=SysComWrite(H1, ADR(Buff[11]), 1, {SYS_INFINITE}10, ADR(PP3));
	WW10b:=SysComWrite(H1, ADR(Buff[12]), 1, {SYS_INFINITE}10, ADR(PP3));
*)
	IF PP3=5// таймаут
		THEN// ошибки
		PP2:= SysComPurge(H1);
		Cnt3:=Cnt3+1;
	END_IF
	


3:
	PP5:=SysComClose(H1);
	// здесь можно сформировать признак ошибки СОМ-порта "ComOpen ERROR"
	ErrorCOM_Mess1:="Com1 Open Error";
	Index:=10;
	
4:
	PP5:=SysComClose(H1);
	// здесь можно сформировать признак ошибки СОМ-порта "ComPurge ERROR"
	ErrorCOM_Mess1:="Com1 Purge Error";
//	Index:=1;// возобновить работу СОМ
	Index:=10;

5:
	PP5:=SysComClose(H1);
	// здесь можно сформировать признак ошибки СОМ-порта "ComWrite ERROR"
	ErrorCOM_Mess1:="Com1 Write Error";
	Index:=1;// возобновить работу СОМ
	
6:
	PP5:=SysComClose(H1);
	// здесь можно сформировать признак ошибки СОМ-порта "ComRead ERROR"
	ErrorCOM_Mess1:="Com1 Read Error";
	Index:=1;// возобновить работу СОМ

7:
	// здесь можно сформировать признак ошибки СОМ-порта "Packet ERROR"
	//	ошибка целостности пакета
	ErrorCOM_Mess1:="Com1 Packet Error";
	Index:=1;// возобновить работу СОМ

10:
	// здесь можно сформировать признак ошибки СОМ-порта
	ErrorCOM_Mess2:="Com1 Can't Open or Close";



150:
		PP2:= SysComPurge(H1);
	Index:=1;


	
END_CASE

END_FUNCTION_BLOCK

// REZERV1/REZ2_1
FUNCTION_BLOCK REZ2_1
VAR CONSTANT
	Timeout_StartOn:TIME:=T#3000MS;//T#10000MS;	
	Timeout_StartTo:TIME:=T#2000MS;//T#3000MS;	
	Timeout_NoPila_Rezerv:TIME:=T#1500MS;//T#3000MS;	
 	Count_PassiveToActive_Other:INT:=15;
END_VAR
VAR_INPUT
	_BMPERR:WORD;// ошибки УСО этого контроллера
	_My_MX_Status:WORD;// входная переменная как MX_Status
	_PilaK_O:WORD;// глоб сетевая посылка из соседнего
	_StatusK_O:WORD;// глоб сетевая посылка из соседнего
	_ReadyK_O:WORD;// глоб сетевая посылка из соседнего
END_VAR
VAR_IN_OUT
	_StateK:RezervState;// Статус контроллера
	_ReadyK:WORD;// Готовность к управлению
	_Cmd_GoPassive:WORD;// команда "Стать пассивным" (от МПУ или из-вне)
END_VAR
VAR_OUTPUT
	_My_MX_Mode:WORD;// выходная переменная как MX_Mode
	_Udo:BOOL:=FALSE;// Вкл/откл U пит +24В на DO
	_MasterOPC:BOOL:=FALSE;// Мастер-переменная ОРС	
	_StateStr:STRING;
	_ReadyStr:WSTRING;
END_VAR
VAR
	NoPila_Rezerv:BOOL;// признак отсутствия пилы соседа
	NoPilaStatus_Rezerv:BOOL;// признак отсутствия пилы Статуса соседа
	NoPilaReady_Rezerv:BOOL;// признак отсутствия пилы Готовность соседа
		NoCOMPila_Rezerv:BOOL;// признак отсутствия пилы соседа через СОМ
		NoCOMPilaStatus_Rezerv:BOOL;// признак отсутствия пилы Статуса соседа через СОМ
		NoCOMPilaReady_Rezerv:BOOL;// признак отсутствия пилы Готовность соседа через СОМ

	Tst1:PilaTst;// функц-блок наличия пилы соседа	
	SetState:SetStateK;// функц-блок установки статуса контролллера	
	PilaStat1:PilaStat;// функц-блок наличия пилы Статуса соседа и самого Статуса
	StatusK_OO:WORD;//статус, выделенный из ПилыСтатуса
	PilaReady1:PilaReady;// функц-блок наличия пилы Готовности соседа и самой Готовности
	ReadyK_OO:WORD;//готовность, выделенная из ПилыГотов

	Tst2:PilaTst;// функц-блок наличия пилы соседа через СОМ	
//	SetState:SetStateK;// функц-блок установки статуса контролллера	
	PilaStat2:PilaStat;// функц-блок наличия пилы Статуса соседа и самого Статуса через СОМ
	StatusK_OOO:WORD;//статус, выделенный из ПилыСтатуса через СОМ
	PilaReady2:PilaReady;// функц-блок наличия пилы Готовности соседа и самой Готовности через СОМ
	ReadyK_OOO:WORD;//готовность, выделенная из ПилыГотов через СОМ
	
	TT1, TT2:TON;
	Cnt_PassiveToActive_Other:INT;

END_VAR

// включить обработку мультиплексора в системе резервирования
{define Use_MX_in_Rezerv}
// отключить обработку мультиплексора в системе резервирования
//{undefine Use_MX_in_Rezerv}

// выдать в окно "Message" подсказку о наличие или отсутствии МХ в проекте и на контроллере
{IF defined (Use_MX_in_Rezerv) }
{info 'MX is present in ELPK'}
{ELSE}
{info 'MX is NOT present in ELPK'}
{END_IF}

CASE _StateK OF
0: _StateStr:='Nothing';
1: _StateStr:='Single';
2: _StateStr:='Active';
3: _StateStr:='Passive';
END_CASE

CASE _ReadyK OF
0: _ReadyStr:="НЕ готов к управлению";
1: _ReadyStr:="Готов к управлению";
END_CASE

IF _BMPERR <> 0
	THEN// есть ошибки УСО - сбросить мою готовность взять управление
	_ReadyK := 0;
	ELSE// нет ошибок УСО - установить мою готовность взять управление
	_ReadyK := 1;
END_IF

// задержка на старте - ничего не делать, пока не отработал таймер
TT1(IN:=1, PT:=Timeout_StartOn{T#10000MS});
IF TT1.Q
	THEN
	// исполняется на старте пока таймер НЕ отработал
	TT2(IN:=1, PT:=Timeout_StartTo{T#3000MS});
	IF (TT2.Q=TRUE) OR (_StateK <> Nothing) 
		THEN
		//
		ELSE	
		Tst1(Pila:=_PilaK_O, TimeOut:=Timeout_NoPila_Rezerv{T#5000MS}, NoPila=>NoPila_Rezerv);
		PilaStat1(PilaStatus:=_StatusK_O, TimeOut:=Timeout_NoPila_Rezerv{T#5000MS}, NoPila=>NoPilaStatus_Rezerv, MyStatus=>StatusK_OO);
		PilaReady1(PilaReady:=_ReadyK_O, TimeOut:=Timeout_NoPila_Rezerv{T#5000MS}, NoPila=>NoPilaReady_Rezerv, MyReady=>ReadyK_OO);

		IF NoPila_Rezerv OR NoPilaStatus_Rezerv OR NoPilaReady_Rezerv
			THEN
			// нет пилы соседа
			SetState(MyState:=Single, StateK=> _StateK, Udo=> _Udo, MasterOPC=> _MasterOPC);
			ELSE
			// есть пила соседа
			IF (StatusK_OO=Active) OR (StatusK_OO=Single)
				THEN
				SetState(MyState:=Passive, StateK=> _StateK, Udo=> _Udo, MasterOPC=> _MasterOPC);
				ELSE
				SetState(MyState:=Active, StateK=> _StateK, Udo=> _Udo, MasterOPC=> _MasterOPC);
			END_IF
		END_IF
	END_IF
	ELSE
	// пока задержка на старте - контролировать пилу, чтобы таймаут вышел (если нет связи)
	Tst1(Pila:=_PilaK_O, TimeOut:=Timeout_NoPila_Rezerv{T#5000MS}, NoPila=>NoPila_Rezerv);	
	PilaStat1(PilaStatus:=_StatusK_O, TimeOut:=Timeout_NoPila_Rezerv{T#5000MS}, NoPila=>NoPilaStatus_Rezerv, MyStatus=>StatusK_OO);
	PilaReady1(PilaReady:=_ReadyK_O, TimeOut:=Timeout_NoPila_Rezerv{T#5000MS}, NoPila=>NoPilaReady_Rezerv, MyReady=>ReadyK_OO);
END_IF

/////////////////   РАБОТА   //////////////////////////////////////////////////////
CASE _StateK OF
Nothing:
Single:	
	Tst1(Pila:=_PilaK_O, TimeOut:=Timeout_NoPila_Rezerv{T#5000MS}, NoPila=>NoPila_Rezerv);
	PilaStat1(PilaStatus:=_StatusK_O, TimeOut:=Timeout_NoPila_Rezerv{T#5000MS}, NoPila=>NoPilaStatus_Rezerv, MyStatus=>StatusK_OO);
	PilaReady1(PilaReady:=_ReadyK_O, TimeOut:=Timeout_NoPila_Rezerv{T#5000MS}, NoPila=>NoPilaReady_Rezerv, MyReady=>ReadyK_OO);

	IF NoPila_Rezerv OR NoPilaStatus_Rezerv OR NoPilaReady_Rezerv
		THEN
		// нет пилы соседа
		SetState(MyState:=Single, StateK=> _StateK, Udo=> _Udo, MasterOPC=> _MasterOPC);
		ELSE
		// есть пила соседа
		IF (StatusK_OO=Passive)
			THEN
			SetState(MyState:=Active, StateK=> _StateK, Udo=> _Udo, MasterOPC=> _MasterOPC);
			ELSIF (StatusK_OO=Active) OR (StatusK_OO=Single)
				THEN	
				SetState(MyState:=Passive, StateK=> _StateK, Udo=> _Udo, MasterOPC=> _MasterOPC);
		END_IF
	END_IF
	_Cmd_GoPassive:=0;//сбросить возможную команду - не должно быть в Single
	{IF defined (Use_MX_in_Rezerv) }
	// если есть 8000 (т.е. сосед отпустил МХ), то можно делать МХ активным
	IF _My_MX_Status.15 = 1
		THEN
		_My_MX_Mode:=8;		
	END_IF
	{END_IF}

Active:
	Tst1(Pila:=_PilaK_O, TimeOut:=Timeout_NoPila_Rezerv{T#5000MS}, NoPila=>NoPila_Rezerv);
	PilaStat1(PilaStatus:=_StatusK_O, TimeOut:=Timeout_NoPila_Rezerv{T#5000MS}, NoPila=>NoPilaStatus_Rezerv, MyStatus=>StatusK_OO);
	PilaReady1(PilaReady:=_ReadyK_O, TimeOut:=Timeout_NoPila_Rezerv{T#5000MS}, NoPila=>NoPilaReady_Rezerv, MyReady=>ReadyK_OO);

	IF NoPila_Rezerv OR NoPilaStatus_Rezerv OR NoPilaReady_Rezerv
		THEN
		// нет пилы соседа
		SetState(MyState:=Single, StateK=> _StateK, Udo=> _Udo, MasterOPC=> _MasterOPC);
		ELSE // есть пила соседа
		IF ReadyK_OO = 1
			THEN// другой контроллер готов взять управление -  проверить мои ошибки УСО
			IF _BMPERR <> 0
				THEN// есть ошибки УСО - сбросить мой признак "Готов к управлению" и перейти в Passive
//				ReadyK := 0;
				SetState(MyState:=Passive, StateK=> _StateK, Udo=> _Udo, MasterOPC=> _MasterOPC);
				ELSE// нет ошибок УСО - установить мой признак "Готов к управлению" и проверить команду "Перейти в Пассив"
//				ReadyK := 1;
				IF _Cmd_GoPassive <> 0
					THEN// есть команда "Перейти в Пассив" - перейти в Passive
					_Cmd_GoPassive:=0;//сбросить команду
					Cnt_PassiveToActive_Other:= Count_PassiveToActive_Other{3};// 3 цикла ждать перехода соседа в Active, не реагируя на его статус
					SetState(MyState:=Passive, StateK=> _StateK, Udo=> _Udo, MasterOPC=> _MasterOPC);
					ELSE// нет команды "Перейти в Пассив" - остаться в Active
					SetState(MyState:=Active, StateK=> _StateK, Udo=> _Udo, MasterOPC=> _MasterOPC);
				END_IF
			END_IF
			ELSE// другой контроллер НЕ готов взять управление - остаться в Active
			SetState(MyState:=Active, StateK=> _StateK, Udo=> _Udo, MasterOPC=> _MasterOPC);
		END_IF
	END_IF
	{IF defined (Use_MX_in_Rezerv) }
	// если есть 8000 (т.е. сосед отпустил МХ), то можно делать МХ активным
	IF _My_MX_Status.15 = 1
		THEN
		_My_MX_Mode:=8;		
	END_IF
	{END_IF}

Passive:
	Tst1(Pila:=_PilaK_O, TimeOut:=Timeout_NoPila_Rezerv{T#5000MS}, NoPila=>NoPila_Rezerv);
	PilaStat1(PilaStatus:=_StatusK_O, TimeOut:=Timeout_NoPila_Rezerv{T#5000MS}, NoPila=>NoPilaStatus_Rezerv, MyStatus=>StatusK_OO);
	PilaReady1(PilaReady:=_ReadyK_O, TimeOut:=Timeout_NoPila_Rezerv{T#5000MS}, NoPila=>NoPilaReady_Rezerv, MyReady=>ReadyK_OO);

///	IF NoPila_Rezerv OR NoPilaStatus_Rezerv OR NoPilaReady_Rezerv
///		THEN
///		// нет пилы соседа
///		SetState(MyState:=Single, StateK=> _StateK, Udo=> _Udo, MasterOPC=> _MasterOPC);
	IF NoPila_Rezerv OR NoPilaStatus_Rezerv OR NoPilaReady_Rezerv
		THEN
		// нет пилы соседа
	{IF defined (Use_MX_in_Rezerv) }
		// MX есть в контроллере - тогда проверяем
		// если есть 8004 (т.е. сосед отпустил МХ или его нет, а я пассивный), то можно установить режим SINGLE
		IF _My_MX_Status = 16#8004
			THEN
			SetState(MyState:=Single, StateK=> _StateK, Udo=> _Udo, MasterOPC=> _MasterOPC);
		END_IF
	{ELSE}
		// MX нет в контроллере - тогда просто установить режим SINGLE
			SetState(MyState:=Single, StateK=> _StateK, Udo=> _Udo, MasterOPC=> _MasterOPC);
	{END_IF}
		ELSE
		// есть пила соседа
		IF (StatusK_OO = Active) OR (StatusK_OO = Single)
			THEN
//			IF BMPERR1 <> 0
//				THEN// есть ошибки УСО - сбросить мою готовность взять управление
//				ReadyK := 0;
//				ELSE// нет ошибок УСО - установить мою готовность взять управление
//				ReadyK := 1;
//			END_IF
			SetState(MyState:=Passive, StateK=> _StateK, Udo=> _Udo, MasterOPC=> _MasterOPC);
			Cnt_PassiveToActive_Other:= 0;
			ELSE
			IF Cnt_PassiveToActive_Other <= 0
				THEN// не надо задержек в реакции
				// сосед не в Active - перейти в Active мне
				SetState(MyState:=Active, StateK=> _StateK, Udo=> _Udo, MasterOPC=> _MasterOPC);
				ELSE
				// счетчик > 0 - только что был переход меня из А в Р - надо ждать пока сосед изменит статус !!!	
				// ждем несколько циклов
				Cnt_PassiveToActive_Other:=Cnt_PassiveToActive_Other-1;
			END_IF
		END_IF
	END_IF
	_Cmd_GoPassive:=0;//сбросить возможную команду - не должно быть в Passive
	{IF defined (Use_MX_in_Rezerv) }
	_My_MX_Mode:=4;
	{END_IF}
	
END_CASE
// Посылать команду в отладочном проекте из визуализации надо в переменную Cmd_GoPassive в виде одной из 1 в слове
//
//
//

END_FUNCTION_BLOCK

// REZERV1/ADDCRC16_1
FUNCTION ADDCRC16_1 : WORD
VAR_INPUT
	X:BYTE;
	_CRC16T:WORD;
END_VAR
VAR
	CRC16_B:BOOL;
	I:INT;
	T:WORD;
END_VAR

FOR I:=1 TO 8 DO
	
	T:=BYTE_TO_WORD(X) XOR _CRC16T;
	IF (T AND 16#1) = 1// если нечетное, то = true
		THEN
		CRC16_B:=TRUE;
		ELSE
		CRC16_B:=FALSE;
	END_IF

	_CRC16T:= SHR(_CRC16T, 1);
	X:= SHR(X,1);
	IF CRC16_B THEN _CRC16T:=_CRC16T XOR 16#A001; END_IF;

END_FOR
ADDCRC16:=_CRC16T;

END_FUNCTION

// K1/std12k5/Ystavki/AutoPNS_YT
	{attribute 'symbol' := 'none'}
FUNCTION_BLOCK AutoPNS_YT EXTENDS Baseobject
VAR_INPUT
	{attribute 'symbol' := 'readwright'}
	Yst_izm:UDINT;
END_VAR
VAR_OUTPUT
	
	{attribute 'symbol' := 'read'}
	Yst:UDINT;
	
END_VAR
VAR
	Yst_Izm_trig:R_TRIG;
	Yst_First_izm:R_TRIG;
	flag:bool;
END_VAR

SUPER^();
Yst_Izm_trig (clk:=((Yst_izm <> Yst) 	AND (Yst_izm >0) AND (Yst_izm < 1000) AND (Yst_izm > Ystavki.YstPNS_YP.Yst)));
IF 	Yst_Izm_trig.Q THEN
	Yst := Yst_izm;
	SaveToFile();
END_IF
Yst_First_izm (clk:=((Yst_izm = 0) AND (Yst = 0) AND flag));
IF	 Yst_First_izm.Q THEN
	Yst := 500;
	Yst_izm := Yst;
	SaveToFile();
END_IF;
flag:=TRUE;

METHOD PROTECTED readPersistent
VAR_INPUT
END_VAR
Yst_izm:=STRING_TO_UDINT(readValue());
END_METHOD

METHOD PROTECTED writePersistent
VAR_INPUT
END_VAR
writeValue(value:= UDINT_TO_STRING(Yst),'Наработка');
END_METHOD

END_FUNCTION_BLOCK

// K2/std12k5/Ystavki/AutoPNS_YT
	{attribute 'symbol' := 'none'}
FUNCTION_BLOCK AutoPNS_YT EXTENDS Baseobject
VAR_INPUT
	{attribute 'symbol' := 'readwright'}
	Yst_izm:UDINT;
END_VAR
VAR_OUTPUT
	
	{attribute 'symbol' := 'read'}
	Yst:UDINT;
	
END_VAR
VAR
	Yst_Izm_trig:R_TRIG;
	Yst_First_izm:R_TRIG;
	flag:bool;
END_VAR

SUPER^();
Yst_Izm_trig (clk:=((Yst_izm <> Yst) 	AND (Yst_izm >0) AND (Yst_izm < 1000) AND (Yst_izm > Ystavki.YstPNS_YP.Yst)));
IF 	Yst_Izm_trig.Q THEN
	Yst := Yst_izm;
	SaveToFile();
END_IF
Yst_First_izm (clk:=((Yst_izm = 0) AND (Yst = 0) AND flag));
IF	 Yst_First_izm.Q THEN
	Yst := 500;
	Yst_izm := Yst;
	SaveToFile();
END_IF;
flag:=TRUE;

METHOD PROTECTED readPersistent
VAR_INPUT
END_VAR
Yst_izm:=STRING_TO_UDINT(readValue());
END_METHOD

METHOD PROTECTED writePersistent
VAR_INPUT
END_VAR
writeValue(value:= UDINT_TO_STRING(Yst),'Наработка');
END_METHOD

END_FUNCTION_BLOCK

// K1/std12k5/Pusk/puskSecond_faza_Chastotny
{attribute 'symbol' := 'none'}
FUNCTION_BLOCK puskSecond_faza_Chastotny EXTENDS StepBySteapAlgoritm
VAR_INPUT
	autoAVOM_canrun_flag:bool;
END_VAR
VAR_OUTPUT
END_VAR
VAR
	{attribute 'symbol' := 'read'}
	timer120:			ph_Timer (table:=ADR(phasesTable)):=		(phaseNumber:=0, delay:=T#120S);
	timer5:				ph_Timer (table:=ADR(phasesTable)):=		(phaseNumber:=2, delay:=T#6S);
	Shup:				CustomPhase (table:=ADR(phasesTable)):=		(phaseNumber:=3);
	Net_Chast:			CustomPhase (table:=ADR(phasesTable)):=		(phaseNumber:=4);
	mvOn:				CustomPhase (table:=ADR(phasesTable)):=		(phaseNumber:=5);
	pGNSmore04:			CustomPhase (table:=ADR(phasesTable)):=		(phaseNumber:=6);
	gotov_K_zagruzke: 	ph_SingleSignal (table:=ADR(phasesTable)):=	(phaseNumber:=7, im:=im.LoadDriveisGranted, expectedValue:=TRUE);

	dPmg_Top:			CustomPhase (table:=ADR(phasesTable)):=		(phaseNumber:=9);
	AutoPNS_Start:		CustomPhase (table:=ADR(phasesTable)):=		(phaseNumber:=10);
END_VAR

SUPER^();
IF 	NOT mvOn.top THEN
	timer120.run (); //запускаем таймер 120 сек
END_IF
IF	(NOT Net_Chast.top) THEN
	timer5.run (); //запускаем таймер 5 сек
END_IF
///////////////////***Команда в ШУП***//////////////////
IF	NOT Shup.start THEN
	Shup.run ();
END_IF
IF	(NOT Shup.top) AND Shup.start THEN
	im.Pusk_SHUP.impulse ();
	Shup.top:=TRUE;
	mvOn.run ();
END_IF
///////////////////***Проверка отсутствия сигнала частотный пуск***//////////////////
IF	 NOT Net_Chast.start THEN
	Net_Chast.run ();
END_IF
IF	Net_Chast.start AND (NOT Net_Chast.top) THEN
	IF	(NOT im.Chastotniy_Pusk.Q) AND (im.Chastotniy_Pusk_CK.status = 1) THEN
		Net_Chast.top:=TRUE;
		timer5.reset ();
	END_IF
END_IF
///////////////////***Проверка отсутствия сигнала неудавшийся частотный пуск***//////////////////
IF	(NOT timer120.top) AND (NOT mvOn.top) THEN
	protections.p_Fail_Chastotniy_Pusk.run();
ELSE
	protections.p_Fail_Chastotniy_Pusk.reset();
END_IF
IF	mvOn.start AND NOT mvOn.top THEN
	IF	(im.mv.onStatus = statusDualInput.STATUS_On) THEN
		mvOn.top:=TRUE;
	END_IF
END_IF
///////////////////////////////////////////////////////
IF 	mvOn.top  THEN 
	IF	NOT pGNSmore04.start AND ((algManager.mode = modegpa.MODE_PUSKPP_Ch) OR (algManager.mode = modegpa.MODE_PUSKAP_Ch)) THEN //проверяем условие по давление за ГНС > 400 кПа
		pGNSmore04.run(); 
	END_IF
	IF	NOT autoAVOM_canrun_flag THEN
		algoritms.S_AutoAVOM.CanRun:=TRUE;
		autoAVOM_canrun_flag:=TRUE;
	END_IF
	timer120.reset ();
	gotov_K_zagruzke.run();
	IF	(NOT dPmg_Top.start) AND ((algManager.mode = modegpa.MODE_PUSKAP_Ch) OR (algManager.mode = modegpa.MODE_PUSKPP_Ch)) THEN
		dPmg_Top.run ();
	END_IF
	protections.p_mvOff.run (); //включаем защиты по МВ и возбудителю
	protections.p_OFFAvarSwitch.run();
	protections.p_RegVozbOff.run();
END_IF;
///////////////////////////////////////////////////////
IF	dPmg_Top.start AND (NOT dPmg_Top.top) THEN
	IF	(NOT im.PerepadDavlenieMasloGaz_Less100.Q) AND (im.PerepadDavlenieMasloGaz_CK.status = 1)AND (ai.PerepadDavlenieMasloGaz.value > 150)	THEN //по аналогу проверяем только значение, т.к. при пуске может уйти в зашкал
		dPmg_Top.top:=TRUE;
		protections.p_PerepadDavlenieMasloGaz.run();
		protections.p_PerepadDavlenieMasloGaz_Less100.run ();
		protections.p_DGazaNaVhodeNagnetatelja_GPA_STOP.reset ();
		protections.p_DGazaNaVyhodeNagnetatelja_GPA_STOP.reset ();
		algoritms.autoNu_2.CanRun:=TRUE;
		algoritms.autoNu_2.run ();
	END_IF
END_IF
///////////////////////////////////////////////////////
IF	pGNSmore04.start AND (NOT pGNSmore04.top) THEN //Давление после ГНС больше 400 кПА
	IF 	(ai.DavlenijaMaslaPosleGNS.interval	>=statusAi.NORMAL) AND (ai.DavlenijaMaslaPosleGNS.value	 > 400) THEN
	  	pGNSmore04.top:=TRUE; 
	END_IF
END_IF
///////////////////////////////////////////////////////
IF	((pGNSmore04.top AND gotov_K_zagruzke.top AND dPmg_Top.top AND ((algManager.mode = modegpa.MODE_PUSKAP_Ch) OR (algManager.mode = modegpa.MODE_PUSKPP_Ch))) OR 
	(gotov_K_zagruzke.top AND ((algManager.mode = modegpa.MODE_PUSKV_Ch) OR (algManager.mode = modegpa.MODE_I)))) AND NOT AutoPNS_Start.top  THEN 
	algoritms.AutoPNS_Start.CanRun :=TRUE;
	algoritms.AutoPNS_Start.run();
	AutoPNS_Start.top:=TRUE;
	end();
END_IF
/////////////////***Запуск АО***///////////////////////////////////////////
IF	(NOT (Net_Chast.top) AND (timer5.top)) OR (timer120.top AND (NOT mvOn.top)) THEN
	algoritms.ao.CanRun:=TRUE;
	algoritms.ao.run ();
END_IF

METHOD PUBLIC run
VAR_INPUT
END_VAR
SUPER^.run();
statusSet.setBit(15,1);
END_METHOD

METHOD PUBLIC reset
VAR_INPUT
END_VAR
SUPER^.reset();
IF	im.mv.onStatus = statusDualInput.STATUS_OFF THEN
	im.Stop_SHUP.impulse ();
END_IF
protections.p_Fail_Chastotniy_Pusk.reset();
statusSet.setBit(15,0);
END_METHOD

END_FUNCTION_BLOCK

// K2/std12k5/Pusk/puskSecond_faza_Chastotny
{attribute 'symbol' := 'none'}
FUNCTION_BLOCK puskSecond_faza_Chastotny EXTENDS StepBySteapAlgoritm
VAR_INPUT
	autoAVOM_canrun_flag:bool;
END_VAR
VAR_OUTPUT
END_VAR
VAR
	{attribute 'symbol' := 'read'}
	timer120:			ph_Timer (table:=ADR(phasesTable)):=		(phaseNumber:=0, delay:=T#120S);
	timer5:				ph_Timer (table:=ADR(phasesTable)):=		(phaseNumber:=2, delay:=T#6S);
	Shup:				CustomPhase (table:=ADR(phasesTable)):=		(phaseNumber:=3);
	Net_Chast:			CustomPhase (table:=ADR(phasesTable)):=		(phaseNumber:=4);
	mvOn:				CustomPhase (table:=ADR(phasesTable)):=		(phaseNumber:=5);
	pGNSmore04:			CustomPhase (table:=ADR(phasesTable)):=		(phaseNumber:=6);
	gotov_K_zagruzke: 	ph_SingleSignal (table:=ADR(phasesTable)):=	(phaseNumber:=7, im:=im.LoadDriveisGranted, expectedValue:=TRUE);

	dPmg_Top:			CustomPhase (table:=ADR(phasesTable)):=		(phaseNumber:=9);
	AutoPNS_Start:		CustomPhase (table:=ADR(phasesTable)):=		(phaseNumber:=10);
END_VAR

SUPER^();
IF 	NOT mvOn.top THEN
	timer120.run (); //запускаем таймер 120 сек
END_IF
IF	(NOT Net_Chast.top) THEN
	timer5.run (); //запускаем таймер 5 сек
END_IF
///////////////////***Команда в ШУП***//////////////////
IF	NOT Shup.start THEN
	Shup.run ();
END_IF
IF	(NOT Shup.top) AND Shup.start THEN
	im.Pusk_SHUP.impulse ();
	Shup.top:=TRUE;
	mvOn.run ();
END_IF
///////////////////***Проверка отсутствия сигнала частотный пуск***//////////////////
IF	 NOT Net_Chast.start THEN
	Net_Chast.run ();
END_IF
IF	Net_Chast.start AND (NOT Net_Chast.top) THEN
	IF	(NOT im.Chastotniy_Pusk.Q) AND (im.Chastotniy_Pusk_CK.status = 1) THEN
		Net_Chast.top:=TRUE;
		timer5.reset ();
	END_IF
END_IF
///////////////////***Проверка отсутствия сигнала неудавшийся частотный пуск***//////////////////
IF	(NOT timer120.top) AND (NOT mvOn.top) THEN
	protections.p_Fail_Chastotniy_Pusk.run();
ELSE
	protections.p_Fail_Chastotniy_Pusk.reset();
END_IF
IF	mvOn.start AND NOT mvOn.top THEN
	IF	(im.mv.onStatus = statusDualInput.STATUS_On) THEN
		mvOn.top:=TRUE;
	END_IF
END_IF
///////////////////////////////////////////////////////
IF 	mvOn.top  THEN 
	IF	NOT pGNSmore04.start AND ((algManager.mode = modegpa.MODE_PUSKPP_Ch) OR (algManager.mode = modegpa.MODE_PUSKAP_Ch)) THEN //проверяем условие по давление за ГНС > 400 кПа
		pGNSmore04.run(); 
	END_IF
	IF	NOT autoAVOM_canrun_flag THEN
		algoritms.S_AutoAVOM.CanRun:=TRUE;
		autoAVOM_canrun_flag:=TRUE;
	END_IF
	timer120.reset ();
	gotov_K_zagruzke.run();
	IF	(NOT dPmg_Top.start) AND ((algManager.mode = modegpa.MODE_PUSKAP_Ch) OR (algManager.mode = modegpa.MODE_PUSKPP_Ch)) THEN
		dPmg_Top.run ();
	END_IF
	protections.p_mvOff.run (); //включаем защиты по МВ и возбудителю
	protections.p_OFFAvarSwitch.run();
	protections.p_RegVozbOff.run();
END_IF;
///////////////////////////////////////////////////////
IF	dPmg_Top.start AND (NOT dPmg_Top.top) THEN
	IF	(NOT im.PerepadDavlenieMasloGaz_Less100.Q) AND (im.PerepadDavlenieMasloGaz_CK.status = 1) AND (ai.PerepadDavlenieMasloGaz.value > 150)	THEN //по аналогу проверяем только значение, т.к. при пуске может уйти в зашкал
		dPmg_Top.top:=TRUE;
		protections.p_PerepadDavlenieMasloGaz.run();
		protections.p_PerepadDavlenieMasloGaz_Less100.run ();
		protections.p_DGazaNaVhodeNagnetatelja_GPA_STOP.reset ();
		protections.p_DGazaNaVyhodeNagnetatelja_GPA_STOP.reset ();
		algoritms.autoNu_2.CanRun:=TRUE;
		algoritms.autoNu_2.run ();
	END_IF
END_IF
///////////////////////////////////////////////////////
IF	pGNSmore04.start AND (NOT pGNSmore04.top) THEN //Давление после ГНС больше 400 кПА
	IF 	(ai.DavlenijaMaslaPosleGNS.interval	>=statusAi.NORMAL) AND (ai.DavlenijaMaslaPosleGNS.value	 > 400) THEN
	  	pGNSmore04.top:=TRUE; 
	END_IF
END_IF
///////////////////////////////////////////////////////
IF	((pGNSmore04.top AND gotov_K_zagruzke.top AND dPmg_Top.top AND ((algManager.mode = modegpa.MODE_PUSKAP_Ch) OR (algManager.mode = modegpa.MODE_PUSKPP_Ch))) OR 
	(gotov_K_zagruzke.top AND ((algManager.mode = modegpa.MODE_PUSKV_Ch) OR (algManager.mode = modegpa.MODE_I)))) AND NOT AutoPNS_Start.top  THEN 
	algoritms.AutoPNS_Start.CanRun :=TRUE;
	algoritms.AutoPNS_Start.run();
	AutoPNS_Start.top:=TRUE;
	end();
END_IF
/////////////////***Запуск АО***///////////////////////////////////////////
IF	(NOT (Net_Chast.top) AND (timer5.top)) OR (timer120.top AND (NOT mvOn.top)) THEN
	algoritms.ao.CanRun:=TRUE;
	algoritms.ao.run ();
END_IF

METHOD PUBLIC reset
VAR_INPUT
END_VAR
SUPER^.reset();
IF	im.mv.onStatus = statusDualInput.STATUS_OFF THEN
	im.Stop_SHUP.impulse ();
END_IF
protections.p_Fail_Chastotniy_Pusk.reset();
statusSet.setBit(15,0);
END_METHOD

METHOD PUBLIC run
VAR_INPUT
END_VAR
SUPER^.run();
statusSet.setBit(15,1);
END_METHOD

END_FUNCTION_BLOCK

// lowLevel_ecl/algoritms/StepBySteapAlgoritm
	{attribute 'symbol' := 'none'}
FUNCTION_BLOCK StepBySteapAlgoritm EXTENDS BaseAlgoritm
VAR_INPUT
	blockIm:BOOL:=true;
END_VAR
VAR_OUTPUT
		{attribute 'symbol' := 'Read'}
	Start:DWORD;
		{attribute 'symbol' := 'Read'}
	Error:DWORD;
		{attribute 'symbol' := 'Read'}
	Top:DWORD;	

END_VAR
VAR

	phasesTable:TableDescriptor;//Пересчитывается только во время работы алгоритма. BaseAlgoritmPhase отрабатываются правильно
	pStart:smartPack:=(status:= Start);
	pError:smartPack:=(status:=Error);
	pTop:smartPack:=(status:= Top);
END_VAR
VAR CONSTANT
END_VAR

SUPER^();
ProcessPhases();

METHOD PUBLIC allPhasesDone : Bool
VAR_INPUT
END_VAR
VAR
	curObject:POINTER TO BaseObject;
	curPhase:IAlgoritmPhase;
END_VAR
curObject:=phasesTable.head;
allPhasesDone:=TRUE;
IF curObject=0 THEN
	RETURN;
END_IF
REPEAT
	IF (__QUERYINTERFACE(curObject^,curPhase)) THEN		
		allPhasesDone:=allPhasesDone AND curPhase.top;			
	END_IF;	
	curObject:=curObject^.getNext();
	UNTIL curObject=0
END_REPEAT
END_METHOD

PROPERTY PUBLIC hasError : bool
GET
hasError:=Error<>0;
END_GET
SET
PROTECTED 
VAR
END_VAR
END_SET
END_PROPERTY

METHOD ProcessPhases : INT
VAR
	curObject:POINTER TO BaseObject;
	curPhase:IAlgoritmPhase;
END_VAR
curObject:=phasesTable.head;
IF curObject=0 THEN
	RETURN;
END_IF
REPEAT
	IF (__QUERYINTERFACE(curObject^,curPhase)) THEN		
			pStart.setBit(bitNum:=curPhase.getPhaseNum(),value:=curPhase.start);
			pError.setBit(bitNum:=curPhase.getPhaseNum(),value:=curPhase.error);
			pTop.setBit(bitNum:=curPhase.getPhaseNum(),value:=curPhase.top);
			curObject^();	
	ELSE
		curObject^();		
	END_IF;
	
	curObject:=curObject^.getNext();
	UNTIL curObject=0
END_REPEAT
END_METHOD

METHOD reset
VAR_INPUT
END_VAR
VAR
	curObject:POINTER TO BaseObject;
	curPhase:IAlgoritmPhase;
END_VAR
SUPER^.reset();

curObject:=phasesTable.head;
IF curObject<>0 THEN
	REPEAT
		curObject^();
		IF (__QUERYINTERFACE(curObject^,curPhase)) THEN		
			curPhase.reset();
			IF blockIm THEN
				curPhase.setBlockIm(FALSE);
			END_IF
		END_IF;
		curObject:=curObject^.getNext();
		UNTIL curObject=0
	END_REPEAT;
END_IF

Start:=0;
Error:=0;
Top:=0;
END_METHOD

METHOD run
VAR_INPUT
END_VAR
VAR
	curObject:POINTER TO BaseObject;
	curPhase:IAlgoritmPhase;
END_VAR
SUPER^.run();
IF blockIm then
	curObject:=phasesTable.head;
	IF curObject=0 THEN
		RETURN;
	END_IF
	REPEAT
		IF (__QUERYINTERFACE(curObject^,curPhase)) THEN		
			curPhase.setBlockIm(TRUE);
		END_IF;
		curObject:=curObject^.getNext();
		UNTIL curObject=0
	END_REPEAT
END_IF
END_METHOD

METHOD PUBLIC writeImStatus
VAR_INPUT
END_VAR
SUPER^.writeImStatus();
END_METHOD

END_FUNCTION_BLOCK

// K1/std12k5/TestIm/BlockIm
FUNCTION BlockIm : BOOL
VAR_INPUT
	im: REFERENCE TO BaseIm;
	block:BOOL;
END_VAR
VAR
END_VAR

IF __ISVALIDREF(im) THEN
	IF block THEN
		im.DisableOpcControl();
	ELSE
		im.EnableOpcControl();
	END_IF
END_IF

END_FUNCTION

// K2/std12k5/TestIm/BlockIm
FUNCTION BlockIm : BOOL
VAR_INPUT
	im: REFERENCE TO BaseIm;
	block:BOOL;
END_VAR
VAR
END_VAR

IF __ISVALIDREF(im) THEN
	IF block THEN
		im.DisableOpcControl();
	ELSE
		im.EnableOpcControl();
	END_IF
END_IF

END_FUNCTION

// lowLevel_ecl/algoritms/phases/BaseAlgoritmPhase
	{attribute 'symbol' := 'none'}
FUNCTION_BLOCK BaseAlgoritmPhase EXTENDS BaseObject
IMPLEMENTS IAlgoritmPhase
VAR_INPUT
	phaseNumber:UINT;
END_VAR
VAR_OUTPUT

END_VAR
VAR
	_start:BOOL;
	_error:BOOL;
	_top:BOOL;
	
	_noImRef:AloneLogMessage();
END_VAR

SUPER^();
IF _start THEN
	IF NOT _top THEN
		_top:=getTop();
		IF NOT _error THEN
			_error:=getError();
		END_IF;
	ELSE
		_error:=FALSE;
	END_IF
END_IF

PROPERTY error : BOOL
GET
error:=_error;
END_GET
END_PROPERTY

METHOD PROTECTED getError : bool
VAR_INPUT
END_VAR
getError:=FALSE;
END_METHOD

METHOD protected GetIm : POINTER TO BaseIm
VAR_INPUT
END_VAR
GetIm:=0;
END_METHOD

METHOD getPhaseNum : UINT
getPhaseNum:=phaseNumber;
END_METHOD

METHOD PROTECTED getTop : bool
VAR_INPUT
END_VAR
getTop:=FALSE;
END_METHOD

METHOD PROTECTED onReset
VAR_INPUT
END_VAR
END_METHOD

METHOD PROTECTED onRun
VAR_INPUT
END_VAR
END_METHOD

METHOD FINAL reset : BOOL
VAR
END_VAR
onReset();

_start:=FALSE;
_error:=FALSE;
_top:=FALSE;
END_METHOD

METHOD FINAL run
VAR
END_VAR
IF NOT _start THEN
	onRun();
	_start:=TRUE;
	_top:=getTop();
	_error:=FALSE;
END_IF
END_METHOD

METHOD setBlockIm
VAR_INPUT
	algRuning	: BOOL;
END_VAR
VAR
	curIm:pointer TO BaseIm;
END_VAR
curIm:=GetIm();
IF curIm<>0 THEN
	IF algRuning THEN
		curIm^.DisableOpcControl();
	ELSE
		curIm^.EnableOpcControl();
	END_IF
ELSE
//	_noImRef.write(CmpLog.LogClass.LOG_ERROR,name,'No Im Ref: ');
END_IF;
END_METHOD

PROPERTY start : BOOL
GET
start:=_start;
END_GET
END_PROPERTY

PROPERTY top : BOOL
GET
top:=_top;
END_GET
END_PROPERTY

END_FUNCTION_BLOCK

// lowLevel_ecl/algoritms/phases/ph_Timer
	{attribute 'symbol' := 'none'}
FUNCTION_BLOCK ph_Timer EXTENDS BaseAlgoritmPhase
VAR_INPUT
	delay:TIME;
	delayParameter:REFERENCE TO TimeParametr;
END_VAR
VAR_OUTPUT
		{attribute 'symbol' := 'read'}
	timer:UINT;
END_VAR
VAR
	_timer:TON;
END_VAR

SUPER^();

_timer(PT:=getDelay());	

timer:=UDINT_TO_UINT(TIME_TO_UDINT(getDelay()-_timer.ET)/1000);

METHOD PROTECTED getDelay : TIME
VAR_INPUT
END_VAR
IF __ISVALIDREF(delayParameter) THEN
	getDelay:=delayParameter.Value;	
ELSE
	getDelay:=delay;	
END_IF
END_METHOD

METHOD PROTECTED getTop : bool
VAR_INPUT
END_VAR
getTop:=_timer.Q;
END_METHOD

METHOD PROTECTED onReset
VAR_INPUT
END_VAR
_timer.IN:=FALSE;
timer:=UDINT_TO_UINT(TIME_TO_UDINT(getDelay())/1000);
END_METHOD

METHOD PROTECTED onRun
VAR_INPUT
END_VAR
_timer.PT:=getDelay();
_timer.IN:=TRUE;
END_METHOD

END_FUNCTION_BLOCK

// lowLevel_ecl/algoritms/phases/CustomPhase
	{attribute 'symbol' := 'none'}
FUNCTION_BLOCK CustomPhase EXTENDS BaseObject
IMPLEMENTS IAlgoritmPhase
VAR_INPUT
	phaseNumber:UINT;
END_VAR
VAR_OUTPUT

END_VAR
VAR
	_start:BOOL;
	_error:BOOL;
	_top:BOOL;
	
	_noImRef:AloneLogMessage();
END_VAR

SUPER^();

METHOD getPhaseNum : UINT
getPhaseNum:=phaseNumber;
END_METHOD

METHOD PROTECTED onReset
VAR_INPUT
END_VAR
END_METHOD

METHOD PROTECTED onRun
VAR_INPUT
END_VAR
END_METHOD

METHOD FINAL reset : BOOL
VAR
END_VAR
onReset();

_start:=FALSE;
_error:=FALSE;
_top:=FALSE;
END_METHOD

METHOD FINAL run
VAR
END_VAR
IF NOT _start THEN
	onRun();
	_start:=TRUE;
	_top:=FALSE;
	_error:=FALSE;
END_IF
END_METHOD

METHOD setBlockIm
VAR_INPUT
	algRuning	: BOOL;
END_VAR
VAR
	curIm:pointer TO BaseIm;
END_VAR
END_METHOD

PROPERTY start : BOOL
GET
start:=_start;
END_GET
SET
_start:=start;
END_SET
END_PROPERTY

PROPERTY top : BOOL
GET
top:=_top;
END_GET
SET
PUBLIC 
VAR
END_VAR
_top:=top;
IF (_top) THEN
	_error:=FALSE;
END_IF
END_SET
END_PROPERTY

PROPERTY error : BOOL
SET
IF NOT (_top) THEN
	_error:=error;
END_IF
END_SET
GET
error:=_error;
END_GET
END_PROPERTY

END_FUNCTION_BLOCK

// lowLevel_ecl/algoritms/phases/ph_SingleSignal
	{attribute 'symbol' := 'none'}
FUNCTION_BLOCK ph_SingleSignal EXTENDS BaseAlgoritmPhase
VAR_INPUT
	Im:REFERENCE TO singleSignal;
	expectedValue:BOOL:=TRUE;
END_VAR
VAR_OUTPUT
END_VAR
VAR
END_VAR

SUPER^();

METHOD PROTECTED getError : bool
VAR_INPUT
END_VAR
getError:=NOT Im.reliability;
END_METHOD

METHOD protected GetIm : POINTER TO BaseIm
VAR_INPUT
END_VAR
GetIm:=adr(Im);
END_METHOD

METHOD PROTECTED getTop : bool
VAR_INPUT
END_VAR
getTop:=(Im.Q=expectedValue) AND (Im.reliability);
END_METHOD

END_FUNCTION_BLOCK

// K1/std12k5/Ystavki/Number_Of_AVOM
	{attribute 'symbol' := 'none'}
FUNCTION_BLOCK Number_Of_AVOM EXTENDS Baseobject
VAR_INPUT
	{attribute 'symbol' := 'readwright'}
	Yst_izm:ARRAY [0..3] OF UINT;
END_VAR
VAR_OUTPUT
	{attribute 'symbol' := 'read'}
	Yst:ARRAY [0..3] OF UINT;
	
END_VAR
VAR
	i:UINT;
	flag:bool;
END_VAR

SUPER^();

FOR i:=0 TO 3 DO
	IF 	(Yst_izm [i] <> Yst [i]) AND NOT (algoritms.Auto_Avom_.isRuning) AND (Yst_izm [i] >=1) AND (Yst_izm [i] <=4) THEN
		Yst[i] := Yst_izm [i];
		SaveToFile();
	END_IF	
	
	IF	(Yst_izm [i] = 0) AND (Yst [i] = 0) AND flag  THEN
		Yst [i] := i+1;
		Yst_izm [i] := Yst [i];
		SaveToFile();
	END_IF;


	
END_FOR;
flag:=true;

METHOD PROTECTED writePersistent
VAR_INPUT
END_VAR

writeValue(value:= UINT_TO_STRING(Yst [0]),'Наработка');
writeValue(value:= UINT_TO_STRING(Yst[1]),'Наработка');
writeValue(value:= UINT_TO_STRING(Yst[2]),'Наработка');
writeValue(value:= UINT_TO_STRING(Yst[3]),'Наработка');
END_METHOD

METHOD PROTECTED readPersistent
VAR_INPUT
END_VAR

Yst_izm [0]:=STRING_TO_UINT(readValue());

Yst_izm [1]:=STRING_TO_UINT(readValue());

Yst_izm [2]:=STRING_TO_UINT(readValue());

Yst_izm [3]:=STRING_TO_UINT(readValue());
END_METHOD

END_FUNCTION_BLOCK

// K2/std12k5/Ystavki/Number_Of_AVOM
	{attribute 'symbol' := 'none'}
FUNCTION_BLOCK Number_Of_AVOM EXTENDS Baseobject
VAR_INPUT
	{attribute 'symbol' := 'readwright'}
	Yst_izm:ARRAY [0..3] OF UINT;
END_VAR
VAR_OUTPUT
	{attribute 'symbol' := 'read'}
	Yst:ARRAY [0..3] OF UINT;
	
END_VAR
VAR
	i:UINT;
	flag:bool;
END_VAR

SUPER^();

FOR i:=0 TO 3 DO
	IF 	(Yst_izm [i] <> Yst [i]) AND NOT (algoritms.Auto_Avom_.isRuning) AND (Yst_izm [i] >=1) AND (Yst_izm [i] <=4) THEN
		Yst[i] := Yst_izm [i];
		SaveToFile();
	END_IF	
	
	IF	(Yst_izm [i] = 0) AND (Yst [i] = 0) AND flag  THEN
		Yst [i] := i+1;
		Yst_izm [i] := Yst [i];
		SaveToFile();
	END_IF;


	
END_FOR;
flag:=true;

METHOD PROTECTED writePersistent
VAR_INPUT
END_VAR

writeValue(value:= UINT_TO_STRING(Yst [0]),'Наработка');
writeValue(value:= UINT_TO_STRING(Yst[1]),'Наработка');
writeValue(value:= UINT_TO_STRING(Yst[2]),'Наработка');
writeValue(value:= UINT_TO_STRING(Yst[3]),'Наработка');
END_METHOD

METHOD PROTECTED readPersistent
VAR_INPUT
END_VAR

Yst_izm [0]:=STRING_TO_UINT(readValue());

Yst_izm [1]:=STRING_TO_UINT(readValue());

Yst_izm [2]:=STRING_TO_UINT(readValue());

Yst_izm [3]:=STRING_TO_UINT(readValue());
END_METHOD

END_FUNCTION_BLOCK

// K1/std12k5/Ystavki/AutoTEN_YP
{attribute 'symbol' := 'none'}
FUNCTION_BLOCK AutoTEN_YP EXTENDS Baseobject
VAR_INPUT
	{attribute 'symbol' := 'readwright'}
	Yst_izm:UINT;
END_VAR
VAR_OUTPUT
	{attribute 'symbol' := 'read'}
	Yst_vkl_TEN:UINT;
	
END_VAR
VAR
	flag:BOOL;
	Yst_Izm_trig:R_TRIG;
	Yst_First_izm:R_TRIG;
END_VAR

SUPER^();
Yst_Izm_trig(clk:=((Yst_izm <> Yst_vkl_TEN) AND (Yst_izm >0) AND (Yst_izm < 100) AND (Yst_izm < Ystavki.Yst_Vykl_TEN.Yst_vykl_TEN)));
IF Yst_Izm_trig.Q  THEN
	Yst_vkl_TEN := Yst_izm;
	SaveToFile();
END_IF
Yst_First_izm(clk:=((Yst_izm = 0) AND (Yst_vkl_TEN = 0) AND flag));
IF	Yst_First_izm.Q THEN
	Yst_vkl_TEN := 25;
	Yst_izm := Yst_vkl_TEN;
	SaveToFile();
END_IF;

flag:=TRUE;

METHOD PROTECTED readPersistent
VAR_INPUT
END_VAR
Yst_izm:=STRING_TO_uint(readValue());
END_METHOD

METHOD PROTECTED writePersistent
VAR_INPUT
END_VAR
writeValue(value:= uint_TO_STRING(Yst_vkl_TEN),'Наработка');
END_METHOD

END_FUNCTION_BLOCK

// K2/std12k5/Ystavki/AutoTEN_YP
{attribute 'symbol' := 'none'}
FUNCTION_BLOCK AutoTEN_YP EXTENDS Baseobject
VAR_INPUT
	{attribute 'symbol' := 'readwright'}
	Yst_izm:UINT;
END_VAR
VAR_OUTPUT
	{attribute 'symbol' := 'read'}
	Yst_vkl_TEN:UINT;
	
END_VAR
VAR
	flag:BOOL;
	Yst_Izm_trig:R_TRIG;
	Yst_First_izm:R_TRIG;
END_VAR

SUPER^();
Yst_Izm_trig(clk:=((Yst_izm <> Yst_vkl_TEN) AND (Yst_izm >0) AND (Yst_izm < 100) AND (Yst_izm < Ystavki.Yst_Vykl_TEN.Yst_vykl_TEN)));
IF Yst_Izm_trig.Q  THEN
	Yst_vkl_TEN := Yst_izm;
	SaveToFile();
END_IF
Yst_First_izm(clk:=((Yst_izm = 0) AND (Yst_vkl_TEN = 0) AND flag));
IF	Yst_First_izm.Q THEN
	Yst_vkl_TEN := 25;
	Yst_izm := Yst_vkl_TEN;
	SaveToFile();
END_IF;

flag:=TRUE;

METHOD PROTECTED readPersistent
VAR_INPUT
END_VAR
Yst_izm:=STRING_TO_uint(readValue());
END_METHOD

METHOD PROTECTED writePersistent
VAR_INPUT
END_VAR
writeValue(value:= uint_TO_STRING(Yst_vkl_TEN),'Наработка');
END_METHOD

END_FUNCTION_BLOCK

// K1/std12k5/Ystavki/AutoTEN_YT
{attribute 'symbol' := 'none'}
FUNCTION_BLOCK AutoTEN_YT EXTENDS Baseobject
VAR_INPUT
		{attribute 'symbol' := 'readwright'}
	Yst_izm:UINT;
END_VAR
VAR_OUTPUT
	{attribute 'symbol' := 'read'}
	Yst_vykl_TEN:UINT;

END_VAR
VAR
	Yst_Izm_trig:R_TRIG;
	Yst_First_izm:R_TRIG;
	flag:bool;
END_VAR

SUPER^();
Yst_Izm_trig(clk:=((Yst_izm <> Yst_vykl_TEN) AND (Yst_izm >0) AND (Yst_izm < 100) AND (Yst_izm > Ystavki.Yst_Vkl_TEN.Yst_vkl_TEN)));
IF Yst_Izm_trig.Q THEN
	Yst_vykl_TEN := Yst_izm;
	SaveToFile();
END_IF
Yst_First_izm(clk:=((Yst_izm = 0) AND (Yst_vykl_TEN = 0 ) AND flag));
IF	Yst_First_izm.Q THEN
	Yst_vykl_TEN := 35;
	Yst_izm := Yst_vykl_TEN;
	SaveToFile();
END_IF;

flag:=TRUE;

METHOD PROTECTED readPersistent
VAR_INPUT
END_VAR
Yst_izm:=STRING_TO_uint(readValue());
END_METHOD

METHOD PROTECTED writePersistent
VAR_INPUT
END_VAR
writeValue(value:= uint_TO_STRING(Yst_vykl_TEN),'Наработка');
END_METHOD

END_FUNCTION_BLOCK

// K2/std12k5/Ystavki/AutoTEN_YT
{attribute 'symbol' := 'none'}
FUNCTION_BLOCK AutoTEN_YT EXTENDS Baseobject
VAR_INPUT
		{attribute 'symbol' := 'readwright'}
	Yst_izm:UINT;
END_VAR
VAR_OUTPUT
	{attribute 'symbol' := 'read'}
	Yst_vykl_TEN:UINT;

END_VAR
VAR
	Yst_Izm_trig:R_TRIG;
	Yst_First_izm:R_TRIG;
	flag:bool;
END_VAR

SUPER^();
Yst_Izm_trig(clk:=((Yst_izm <> Yst_vykl_TEN) AND (Yst_izm >0) AND (Yst_izm < 100) AND (Yst_izm > Ystavki.Yst_Vkl_TEN.Yst_vkl_TEN)));
IF Yst_Izm_trig.Q THEN
	Yst_vykl_TEN := Yst_izm;
	SaveToFile();
END_IF
Yst_First_izm(clk:=((Yst_izm = 0) AND (Yst_vykl_TEN = 0 ) AND flag));
IF	Yst_First_izm.Q THEN
	Yst_vykl_TEN := 35;
	Yst_izm := Yst_vykl_TEN;
	SaveToFile();
END_IF;

flag:=TRUE;

METHOD PROTECTED readPersistent
VAR_INPUT
END_VAR
Yst_izm:=STRING_TO_uint(readValue());
END_METHOD

METHOD PROTECTED writePersistent
VAR_INPUT
END_VAR
writeValue(value:= uint_TO_STRING(Yst_vykl_TEN),'Наработка');
END_METHOD

END_FUNCTION_BLOCK

// K1/std12k5/Narabotka/Avom1
	{attribute 'symbol' := 'none'}
FUNCTION_BLOCK Avom1 EXTENDS Vent
VAR_INPUT
END_VAR
VAR_OUTPUT
		{attribute 'symbol' := 'read'}
	narabotka:UDINT;
	narabotka_:ExtNarabotka (table:=ADR (objectTable)):=(saveInterval:=T#1H);
END_VAR
VAR
	(*timer:RTC;	
	saveTimer:TON:=(PT:=T#600S);
	Narabotka_hour:R_TRIG;
	AvomStartted:R_TRIG;
	narabotka_Izm:UDINT;*)
END_VAR

SUPER^();
narabotka_.started:=onstatus=statusDualInput.STATUS_ON;
narabotka:=(narabotka_.narabotka/3600);
(*
AvomStartted(CLK:=im.v1_Avom.onStatus=statusDualInput.status_on);

	timer.PDT:=UDINT_TO_DT(narabotka_izm);

IF im.v1_Avom.onStatus=statusDualInput.status_on THEN
	narabotka_izm:=DT_TO_UDINT( timer.CDT);
	timer.EN:=TRUE;
ELSE
	timer.EN:=FALSE;
END_IF
narabotka_hour (clk:=(narabotka_izm >=3600));
IF	narabotka_hour.Q THEN
	narabotka:=narabotka+1;
	timer.EN:=FALSE;
	narabotka_izm:=0;
END_IF
timer();

saveTimer(IN:=true);
IF saveTimer.Q THEN
	SaveToFile();
	saveTimer(IN:=FALSE);
END_IF*)

METHOD PROTECTED readPersistent
VAR_INPUT
END_VAR

narabotka:=STRING_TO_UDINT(readValue());
narabotka_izm:=STRING_TO_UDINT(readValue());
END_METHOD

METHOD PROTECTED writePersistent
VAR_INPUT
END_VAR

writeValue(value:= UDINT_TO_STRING(narabotka),'Наработка');
writeValue(value:= UDINT_TO_STRING(narabotka_izm),'Наработка_izm');
END_METHOD

END_FUNCTION_BLOCK

// K2/std12k5/Natabotka/Avom1
	{attribute 'symbol' := 'none'}
FUNCTION_BLOCK Avom1 EXTENDS Vent
VAR_INPUT
END_VAR
VAR_OUTPUT
		{attribute 'symbol' := 'read'}
	narabotka:UDINT;
	
	narabotka_:ExtNarabotka (table:=ADR (objectTable)):=(saveInterval:=T#1H);
END_VAR
VAR
(*	timer:RTC;	
	saveTimer:TON:=(PT:=T#600S);
	Narabotka_hour:R_TRIG;
	AvomStartted:R_TRIG;
	narabotka_Izm:UDINT;*)
END_VAR

SUPER^();
narabotka_.started:=onstatus=statusDualInput.STATUS_ON;
narabotka:=(narabotka_.narabotka/3600);
(*
AvomStartted(CLK:=im.v1_Avom.onStatus=statusDualInput.status_on);

	timer.PDT:=UDINT_TO_DT(narabotka_izm);

IF im.v1_Avom.onStatus=statusDualInput.status_on THEN
	narabotka_izm:=DT_TO_UDINT( timer.CDT);
	timer.EN:=TRUE;
ELSE
	timer.EN:=FALSE;
END_IF
narabotka_hour (clk:=(narabotka_izm >=3600));
IF	narabotka_hour.Q THEN
	narabotka:=narabotka+1;
	timer.EN:=FALSE;
	narabotka_izm:=0;
END_IF
timer();

saveTimer(IN:=true);
IF saveTimer.Q THEN
	SaveToFile();
	saveTimer(IN:=FALSE);
END_IF*)

METHOD PROTECTED readPersistent
VAR_INPUT
END_VAR

narabotka:=STRING_TO_UDINT(readValue());
narabotka_izm:=STRING_TO_UDINT(readValue());
END_METHOD

METHOD PROTECTED writePersistent
VAR_INPUT
END_VAR

writeValue(value:= UDINT_TO_STRING(narabotka),'Наработка');
writeValue(value:= UDINT_TO_STRING(narabotka_izm),'Наработка_izm');
END_METHOD

END_FUNCTION_BLOCK

// lowLevel_ecl/im/ventvs/Vent
	{attribute 'symbol' := 'none'}
FUNCTION_BLOCK Vent EXTENDS Ventvs
VAR_INPUT
END_VAR
VAR_OUTPUT
END_VAR
VAR
END_VAR

SUPER^();

END_FUNCTION_BLOCK

// lowLevel_ecl/im/ventvs/Ventvs
	{attribute 'symbol' := 'none'}
FUNCTION_BLOCK PUBLIC Ventvs EXTENDS DualStateSwitch;
VAR_INPUT
	inLocal: REFERENCE TO ReliableBit;	
	inDistance: REFERENCE TO ReliableBit;
	inAuto:REFERENCE TO ReliableBit;
	inManual: REFERENCE TO ReliableBit;
	inBreakCmdOn: REFERENCE TO ReliableBit;
	inBreakCmdOff:REFERENCE TO ReliableBit;	
	
	inErrorOverloud: REFERENCE TO ReliableBit;	
	inErrorPowerOff: REFERENCE TO ReliableBit;
	inErrorBlock: REFERENCE TO ReliableBit;	
END_VAR
VAR_OUTPUT
	local: BOOL;	
	distance: BOOL;
	errorOverloud: BOOL;	
	errorPowerOff: BOOL;
	errorBlock: BOOL;
	auto:BOOL;
	manual:BOOL;
	breakCmdOn: BOOL;
	breakCmdOff:BOOL;		
END_VAR
VAR
	outputsSets:TOF:=(PT:=T#3S);
END_VAR

SUPER^();

local:=checkArg(inLocal);	
distance:=checkArg(inDistance);
errorOverloud:=checkArg(inErrorOverloud);	
errorPowerOff:=checkArg(inErrorPowerOff);
errorBlock:=checkArg(inErrorBlock);
auto:=checkArg(inAuto);
manual:=checkArg(inManual);

outputsSets(in:=validAndTrue(input:=CmdOn) OR validAndTrue(input:=CmdOff));
breakCmdOn:=checkArg(inBreakCmdOn)AND NOT (outputsSets.Q);
breakCmdOff:=checkArg(inBreakCmdOff)AND NOT (outputsSets.Q);

PROPERTY PUBLIC lastComandIsOn : bool
GET
lastComandIsOn:=_lastCmd=statusDualInput.STATUS_ON;
END_GET
END_PROPERTY

METHOD PROTECTED getSdvig : BOOL
VAR_INPUT
END_VAR
getSdvig:=FALSE;
IF (NOT Local) THEN
	getSdvig:=super^.getSdvig();
END_IF
END_METHOD

METHOD public writeImStatus
VAR_INPUT
END_VAR
SUPER^.writeImStatus();

statusSet.setBit(5,local);
statusSet.setBit(6,distance);
statusSet.setBit(7,auto);
statusSet.setBit(8,manual);
statusSet.setBit(9,errorOverloud);
statusSet.setBit(10,errorPowerOff);
statusSet.setBit(11,errorBlock);
statusSet.setBit(12,breakCmdOn);
statusSet.setBit(13,breakCmdOff);

statusSet.setBit(14,lastComandIsOn);
END_METHOD

END_FUNCTION_BLOCK

// K1/std12k5/Narabotka/Avom2
	{attribute 'symbol' := 'none'}
FUNCTION_BLOCK Avom2 EXTENDS Vent
VAR_INPUT
END_VAR
VAR_OUTPUT
		{attribute 'symbol' := 'read'}
	narabotka:UDINT;
	narabotka_:ExtNarabotka (table:=ADR (objectTable)):=(saveInterval:=T#1H);
END_VAR
VAR
	(*timer:RTC;	
	saveTimer:TON:=(PT:=T#600S);
	Narabotka_hour:R_TRIG;
	AvomStartted:R_TRIG;
	narabotka_Izm:UDINT;*)
END_VAR

SUPER^();
narabotka_.started:=onstatus=statusDualInput.STATUS_ON;
narabotka:=(narabotka_.narabotka/3600);
(*
AvomStartted(CLK:=im.v2_Avom.onStatus=statusDualInput.status_on);

	timer.PDT:=UDINT_TO_DT(narabotka_izm);

IF im.v2_Avom.onStatus=statusDualInput.status_on THEN
	narabotka_izm:=DT_TO_UDINT( timer.CDT);
	timer.EN:=TRUE;
ELSE
	timer.EN:=FALSE;
END_IF
narabotka_hour (clk:=(narabotka_izm >=3600));
IF	narabotka_hour.Q THEN
	narabotka:=narabotka+1;
	timer.EN:=FALSE;
	narabotka_izm:=0;
END_IF
timer();

saveTimer(IN:=true);
IF saveTimer.Q THEN
	SaveToFile();
	saveTimer(IN:=FALSE);
END_IF*)

METHOD PROTECTED readPersistent
VAR_INPUT
END_VAR

narabotka:=STRING_TO_UDINT(readValue());
narabotka_izm:=STRING_TO_UDINT(readValue());
END_METHOD

METHOD PROTECTED writePersistent
VAR_INPUT
END_VAR

writeValue(value:= UDINT_TO_STRING(narabotka),'Наработка');
writeValue(value:= UDINT_TO_STRING(narabotka_izm),'Наработка_izm');
END_METHOD

END_FUNCTION_BLOCK

// K2/std12k5/Natabotka/Avom2
	{attribute 'symbol' := 'none'}
FUNCTION_BLOCK Avom2 EXTENDS Vent
VAR_INPUT
END_VAR
VAR_OUTPUT
		{attribute 'symbol' := 'read'}
	narabotka:UDINT;
	
	narabotka_:ExtNarabotka (table:=ADR (objectTable)):=(saveInterval:=T#1H);
END_VAR
VAR
	(*timer:RTC;	
	saveTimer:TON:=(PT:=T#600S);
	Narabotka_hour:R_TRIG;
	AvomStartted:R_TRIG;
	narabotka_Izm:UDINT;*)
END_VAR

SUPER^();
narabotka_.started:=onstatus=statusDualInput.STATUS_ON;
narabotka:=(narabotka_.narabotka/3600);
(*
AvomStartted(CLK:=im.v2_Avom.onStatus=statusDualInput.status_on);

	timer.PDT:=UDINT_TO_DT(narabotka_izm);

IF im.v2_Avom.onStatus=statusDualInput.status_on THEN
	narabotka_izm:=DT_TO_UDINT( timer.CDT);
	timer.EN:=TRUE;
ELSE
	timer.EN:=FALSE;
END_IF
narabotka_hour (clk:=(narabotka_izm >=3600));
IF	narabotka_hour.Q THEN
	narabotka:=narabotka+1;
	timer.EN:=FALSE;
	narabotka_izm:=0;
END_IF
timer();

saveTimer(IN:=true);
IF saveTimer.Q THEN
	SaveToFile();
	saveTimer(IN:=FALSE);
END_IF*)

METHOD PROTECTED readPersistent
VAR_INPUT
END_VAR

narabotka:=STRING_TO_UDINT(readValue());
narabotka_izm:=STRING_TO_UDINT(readValue());
END_METHOD

METHOD PROTECTED writePersistent
VAR_INPUT
END_VAR

writeValue(value:= UDINT_TO_STRING(narabotka),'Наработка');
writeValue(value:= UDINT_TO_STRING(narabotka_izm),'Наработка_izm');
END_METHOD

END_FUNCTION_BLOCK

// K1/std12k5/Narabotka/Avom3
	{attribute 'symbol' := 'none'}
FUNCTION_BLOCK Avom3 EXTENDS Vent
VAR_INPUT
END_VAR
VAR_OUTPUT
		{attribute 'symbol' := 'read'}
	narabotka:UDINT;
	narabotka_:ExtNarabotka (table:=ADR (objectTable)):=(saveInterval:=T#1H);
END_VAR
VAR
	(*timer:RTC;	
	saveTimer:TON:=(PT:=T#600S);
	Narabotka_hour:R_TRIG;
	AvomStartted:R_TRIG;
	narabotka_Izm:UDINT;*)
END_VAR

SUPER^();
narabotka_.started:=onstatus=statusDualInput.STATUS_ON;
narabotka:=(narabotka_.narabotka/3600);
(*
AvomStartted(CLK:=im.v3_Avom.onStatus=statusDualInput.status_on);

	timer.PDT:=UDINT_TO_DT(narabotka_izm);

